# B&R Automation Studio project TD52 (part 131)

#### VisOPCyclic.st - Visualisation Communication Cyclic
```iecst
(*******************************************************************************
VisOP	 			 VISU and bus coupling variables

This code is confidential and proprietary to the INNIO Company.
It may not be used in any form, or reproduced in any manner,
without written permission of the INNIO Company.
Copyright, INNIO Company, 2023

Customized modifications: -
------------------------

History:
-------
V0.1.0	13.09.2012	Graus		new
V0.1.1	23.04.2013	Graus		MM2VIS.rP_Set_Min in AUTO and TEST to Para-value, otherwise is 0
V4.00.0 11.02.2014 	Graus,		change Version TO 4.0
V4.00.1	19.02.2014 zengerer		iIdx_OMSS, iIdx_RSS changed to DINT because of OPC UA troubles
V4.00.2 05.03.2014 	Graus,		add progress indication OF engine operation FOR VIS (iSt_VIS_Porgress)
V4.00.3 14.03.2014 	Graus,		add bEng_Rdy_Aut to MM2VIS structure and assign it for visualization
V4.01.0 19.05.2014  Denk		IN_OP.rP_RedDI_EU_Norm changed
V4.02.0 02.07.2014  Graus,		add MM2VIS.bP_Red_Sp_Lim1Act, 2 and 3
V4.02.1	15.10.2014	Caks,		added glow ignition power reduction
V4.02.2	17.02.2015	Graus,		add visu interface for power reduction by hierarchy controller
V4.02.3	04.05.2015	Denk,		add visu interfaces for OPC
V4.04.0	08.07.2016	Zengerer	BETA: Step Time Display Information
		17.11.2016	Gomez Ortiz	Addition of B2168 generator air inlet temperature power reduction
		21.12.2016  Denk		Modification for WinMOD simulation
V4.05.0 14.06.2017	Gomez Ortiz Addition of power limitation due to low engine cooling water temperature, Spec_Start_Load_release_manual_start.doc
V4.05.0 19.10.2017  Gomez Ortiz Addition of bImp_UnitOpHour to the MM2VIS struct
		24.10.2017	Zingerle	SWAT 920 Rel.5, power reduction with difference pressure minimum
		21.01.2018	Perktold,	hardware operation mode switch added
V4.07.0	11.10.2018	lettenb.	Di: tF_N_DI_Inc/Dec added for diagnosis
V4.07.4	29.03.2019	Hohensinner	Bugfixing: added missing interface to VIS for PRed CppInt
		26.04.2019	Hohensinner	Set minimum time for speed pulses for HMI to 2sec
V4.10.0 10.12.2020  Zuschnig	Included power reduction for Tecjet differential pressure
		18.01.2021	Perktold	included spec. gas p.red in MM2VIS
		25.01.2021	Zuschnig	Change MM2VIS.P_UNRED from Norm to kW
V4.11.0	20.08.2021 	Keller		Add Messages bMsg9057 - bMsg9060
		22.11.2021	Perktold,	added myPlant Remote Status computation
		22.12.2021	Andre		added Power reduction by CAN communication failure for half or more SAFI or too many SAFI reboots
V4.12.0	12.01.2023	Tinello		Deleted power reduction by T1HP / Added power reduction by T2HP and T2LP
		22.01.2023  Zuschnig	Include power reduction H2 content
		24.03.2023	Perktold	Write on PRed-MM2VIS variables just when ParaSetupOk is true - mitigation for wrong values on HMI
V4.13.0	05.07.2023	Zuschnig	Removed Step Time Display Information
  		26.01.2024 	Zuschnig 	Split of power reduction FPR

Instructions for use:
--------------------

Outstandings:
------------

(*******************************************************************************)

PROGRAM _CYCLIC

	(* Output: MM2VIS *)
	(* myPlant Remote Status computation *)
	IF bParaSetupOk_2s AND NOT bGnlTrip AND NOT bRequest_Bloc AND NOT OUT_OP.bEng_Bloc AND bOMSS_AUTO AND bRSS_REM AND (IN_OP.iIdx_SyOMSS = 2) AND Para.bRemoteReqMyPlantActive THEN
		MM2VIS.iMyPlant_Remote_Ready		:= 2;
	ELSE
		(* Reset myPlant demand in following cases, trip, engine blocking active, engine not in AUTO + REMOTE mode or function not active*)
		IF VIS2MM.bRemoteReq_myPlant THEN
			VIS2MM.bRemoteReq_myPlant 		:= FALSE;
		END_IF;
		IF Para.bRemoteReqMyPlantActive THEN
			MM2VIS.iMyPlant_Remote_Ready	:= 1;
		ELSE
			MM2VIS.iMyPlant_Remote_Ready	:= 0;
		END_IF;
	END_IF;

	MM2VIS.M_ANF := 			M_ANF;
	MM2VIS.iSt_OpMode_Main := 	iSt_OpMode_Main;
	MM2VIS.rN_Set := 			OUT_OP.rN_Set_Norm * Para.rN_EngNom;
	MM2VIS.rP_Act_Filt := 		OUT_OP.rP_Act_Norm_Filt * OUT_OP.rP_Nom;
	MM2VIS.rP_Set := 			OUT_OP.rP_Set_Norm * OUT_OP.rP_Nom;
	MM2VIS.P_UNRED := 			OUT_OP.rP_Set_Unred_Norm * OUT_OP.rP_Nom;

	MM2VIS.bP_Red_Active := 	OUT_OP.bP_Red_Active OR xTP_bP_Red_Active.Q;
	xTP_bP_Red_Active(IN := 	MM2VIS.bP_Red_Active, PT := T#1s);				(*min 1s TRUE to mitigate wrong values on HMI*)

	MM2VIS.RedPower := 			RedPower_Norm * OUT_OP.rP_Nom;
	MM2VIS.iIdx_Eng_State := 	iIdx_Eng_State;
	MM2VIS.iIdx_Pred_Type := 	OUT_OP.iIdx_Pred_Type;
	MM2VIS.iSt_OpMode_Sub := 	iSt_OpMode_Sub;
	MM2VIS.iSt_OpMode_Deg := 	iSt_OpMode_Deg;
	MM2VIS.bMsg2125 := 		bMsg2125;
	MM2VIS.bMsg2126 := 		bMsg2126;
	MM2VIS.bMsg2127 := 		bMsg2127;
	MM2VIS.bMsg2128 := 		bMsg2128;
	MM2VIS.bMsg2129 := 		bMsg2129;
	MM2VIS.bMsg2130 := 		bMsg2130;
	MM2VIS.bMsg2131 := 		bMsg2131;
	MM2VIS.bMsg2132 := 		bMsg2132;
	MM2VIS.bMsg2143 := 		bMsg2143;
	MM2VIS.bMsg2144 := 		bMsg2144;
	MM2VIS.bMsg2146 := 		bMsg2146;
	MM2VIS.bMsg2147 := 		bMsg2147;
	MM2VIS.bMsg2148 := 		bMsg2148;
	MM2VIS.bMsg2149 := 		bMsg2149;
	MM2VIS.bMsg2150 := 		bMsg2150;
	MM2VIS.bMsg2152 := 		bMsg2152;
	MM2VIS.bMsg2153 :=		bMsg2153;
	MM2VIS.bMsg2154 :=		bMsg2154;
	MM2VIS.bMsg2155 :=		bMsg2155;
	MM2VIS.bMsg2158 :=		bMsg2158;
	MM2VIS.bMsg2159 :=		bMsg2159;
	MM2VIS.bMsg2160 :=		bMsg2160;
	MM2VIS.bMsg2161 :=		bMsg2161;
	MM2VIS.bMsg2163 :=		bMsg2163;
	MM2VIS.bMsg2164 :=		bMsg2164;
	MM2VIS.bMsg2803 :=		bMsg2803;
	MM2VIS.bMsg3229 :=		bMsg3229;
	MM2VIS.bMsg3230 :=		bMsg3230;
	MM2VIS.bMsg3231 :=		bMsg3231;
	MM2VIS.bMsg2140 :=		bMsg2140;
	MM2VIS.bMsg3506 :=		bMsg3506;
	MM2VIS.bMsg2082 :=		bMsg2082;
	MM2VIS.bMsg1188 :=		bMsg1188;
	MM2VIS.bMsg2097 :=		bMsg2097;
	MM2VIS.bMsg1108 :=		bMsg1108;
	MM2VIS.bEng_RPSDem :=		OUT_OP.bEng_RPSDem;
	MM2VIS.bEng_Rdy_Aut_Exc :=	OUT_OP.bEng_Rdy_Aut_Exc;
	MM2VIS.rP_Ramp_IncGrad_All_Norm := OUT_OP.rP_Ramp_IncGrad_All_Norm;
	MM2VIS.rP_Ramp_DecGrad_All_Norm := OUT_OP.rP_Ramp_DecGrad_All_Norm;

	MM2VIS.bMsg1225 :=	bMsg1225;
	MM2VIS.bMsg1226 :=	bMsg1226;
	MM2VIS.bMsg1227 :=	bMsg1227;
	MM2VIS.bMsg1228 :=	bMsg1228;
	MM2VIS.bMsg1229 :=	bMsg1229;
	MM2VIS.bMsg1230 :=	bMsg1230;
	MM2VIS.bMsg1231 :=	bMsg1231;
	MM2VIS.bMsg1232 :=	bMsg1232;
	MM2VIS.bMsg1233 :=	bMsg1233;
	MM2VIS.bMsg1234 :=	bMsg1234;
	MM2VIS.bMsg1237 :=	bMsg1237;
	MM2VIS.bMsg1238 :=	bMsg1238;
	MM2VIS.bMsg1241 :=	bMsg1241;
	MM2VIS.bMsg1242 :=	bMsg1242;
	MM2VIS.bMsg1243 :=	bMsg1243;
	MM2VIS.bMsg1244 :=	bMsg1244;

	MM2VIS.bMsg2170 :=	bMsg2170;
	MM2VIS.bMsg2936 :=	bMsg2936;

	(* from HAL IO *)
	(* to HAL IO *)
	MM2VIS.bEng_Aux_Dem_CDR :=	OUT_OP.tEng_Aux_Dem_CDR.Do;
	MM2VIS.bEng_Run :=			OUT_OP.tEng_Run.Do;

	(* Input: VIS2MM *)
	bStart := 			VIS2MM.bStart;
	VIS2MM.bStart := 	FALSE;	(* reset VIS button *)
	bStop := 			VIS2MM.bStop;
	VIS2MM.bStop := 	FALSE;	(* reset VIS button *)

	(* HARDWARE OPERATION MODE SWITCHES *)
	IF IN_OP.tHW_Switches.bGoodQual THEN
		OUT_OP.iIdx_OMSS			:= IN_OP.tHW_Switches.iIdx_OMS_Hw;
		OUT_OP.iIdx_RSS 			:= IN_OP.tHW_Switches.iIdx_RMS_Hw;
		VIS2MM.iIdx_OMSS			:= INT_TO_DINT(IN_OP.tHW_Switches.iIdx_OMS_Hw);
		VIS2MM.iIdx_RSS				:= INT_TO_DINT(IN_OP.tHW_Switches.iIdx_RMS_Hw);
		MM2VIS.bDont_show_switches	:= TRUE;	(* DON'T show switches on HMI *)
	ELSE	(* OPERATION MODE SWITCHES ON HMI *)
		OUT_OP.iIdx_OMSS 			:= DINT_TO_INT(VIS2MM.iIdx_OMSS);
		OUT_OP.iIdx_RSS 			:= DINT_TO_INT(VIS2MM.iIdx_RSS);
		MM2VIS.bDont_show_switches	:= FALSE;	(* show switches on HMI *)
	END_IF;

	OUT_OP.bStart	:= 	bStart;		(* to AuxiliariesGeneral starter tasks *)
	OUT_OP.bStop	:= 	bStop;		(* to AuxiliariesGeneral starter tasks *)

	MM2VIS.bMainMode_Idle := xOpMode.Idle;
	MM2VIS.bMainMode_Grid := xOpMode.NetP;
	MM2VIS.bMainMode_Island := xOpMode.Island;

	xTON_ParaOK_1s(IN := IN_OP.tPB2MM.bParaSetupOk, PT := T#1s);	(*Delay to mitigate wrong values on HMI*)
	IF xTON_ParaOK_1s.Q THEN

		MM2VIS.rP_Nom			:=		OUT_OP.rP_Nom;

		MM2VIS.rP_RedDelta_Knck_Norm		:= 1.0 - IN_OP.rP_Red_Knck_Norm;
		MM2VIS.rP_RedDelta_Ch_T2s_Norm		:= 1.0 - IN_OP.rP_Red_Ch_T2s_Norm_TC5;
		MM2VIS.rP_RedDelta_Misf_Norm		:= 1.0 - IN_OP.rP_Red_Misf_Norm;
		MM2VIS.rP_RedDelta_EGT_Norm			:= 1.0 - IN_OP.rP_Red_EGT_Norm;
		MM2VIS.rP_RedDelta_T_InAirER_Norm	:= 1.0 - IN_OP.rP_Red_T_InAirER_Norm;
		MM2VIS.rP_RedDelta_Leanox_Norm		:= 1.0 - IN_OP.rP_Red_Leanox_Norm;
		MM2VIS.rP_RedDelta_CH4_Norm			:= 1.0 - IN_OP.rP_Red_CH4_Norm;
		MM2VIS.rP_RedDelta_GasPr_Norm		:= 1.0 - IN_OP.rP_Red_GasPr_Norm;
		MM2VIS.rP_RedDelta_SuctPr_Norm		:= 1.0 - IN_OP.rP_Red_SuctPr_Norm;
		MM2VIS.rP_RedDelta_TC_Norm			:= 1.0 - IN_OP.rP_Red_TC_Norm;
		MM2VIS.rP_RedDelta_T_HWR_Norm		:= 1.0 - IN_OP.rP_Red_T_HWR_Norm;
		MM2VIS.rP_RedDelta_T_ECW_Norm		:= 1.0 - IN_OP.rP_Red_T_ECW_Norm;
		MM2VIS.rP_RedDelta_T_Oil_Norm		:= 1.0 - IN_OP.rP_Red_T_Oil_Norm;
		MM2VIS.rP_RedDelta_Pr_PCGT_Norm		:= 1.0 - IN_OP.rP_Red_Pr_PCGT_Norm;
		MM2VIS.rP_RedDelta_CosPCtr_U_Norm 	:= 1.0 - IN_OP.rP_Red_CosPCtr_U_Norm;
		MM2VIS.rP_RedDelta_CosPCtr_F_Norm 	:= 1.0 - IN_OP.rP_Red_CosPCtr_F_Norm;
		MM2VIS.rP_RedDelta_CosPCtr_T_Norm 	:= 1.0 - IN_OP.rP_Red_CosPCtr_T_Norm;
		MM2VIS.rP_RedDelta_Sp_Lim1_Norm		:= 1.0 - IN_OP.rP_Red_Sp_Lim1_Norm;
		MM2VIS.rP_RedDelta_Sp_Lim2_Norm		:= 1.0 - IN_OP.rP_Red_Sp_Lim2_Norm;
		MM2VIS.rP_RedDelta_Sp_Lim3_Norm		:= 1.0 - IN_OP.rP_Red_Sp_Lim3_Norm;
		MM2VIS.rP_RedDelta_EVU_Norm			:= 1.0 - IN_OP.rP_RedDI_EU_Norm;
		MM2VIS.rP_RedDelta_AI_Norm			:= 1.0 - IN_OP.rP_Red_AI_Norm;
		MM2VIS.rP_RedDelta_ExtBus_Norm		:= 1.0 - IN_OP.rP_Red_ExtBus_Norm;
		MM2VIS.rP_RedDelta_Hum_Norm			:= 1.0 - IN_OP.rP_Red_Hum_Norm;
		MM2VIS.rP_RedDelta_PBC_Norm 		:= 1.0 - IN_OP.rP_Red_PBC_Norm;
		MM2VIS.rP_RedDelta_Knck_Opti_Norm	:= 1.0 - IN_OP.rP_Red_Knck_Opti_Norm;
		MM2VIS.rP_RedDelta_SG_Norm			:= 1.0 - MIN(IN_OP.rP_Red_SG_Norm_Pred, IN_OP.rP_Red_SG_Norm_FPR);
		MM2VIS.rP_RedDelta_Pr_CC_Norm		:= 1.0 - IN_OP.rP_Red_Pr_CC_Norm;
		MM2VIS.rP_RedDelta_HiCtr_Norm		:= 1.0 - IN_OP.rP_Red_HiCtr_Norm;
		MM2VIS.rP_RedDelta_T_Transformer_Norm		:= 1.0 - IN_OP.rP_Red_TransformerWarning_Norm;
		MM2VIS.rP_RedDelta_T_GenSwitchCab_Norm		:= 1.0 - IN_OP.rP_Red_TempMax_GenCB_Norm;
		MM2VIS.rP_RedDelta_T_GenAirIn_Norm	:= 1.0 - IN_OP.rP_Red_T_GenAirIn_Norm;
		MM2VIS.rP_RedDelta_Pr_GR_Norm		:= 1.0 - IN_OP.rP_Red_Pr_GR_Norm;
		MM2VIS.rP_RedDelta_CppInt_Norm		:= 1.0 - IN_OP.rP_Red_CppInt_Norm;
		MM2VIS.rP_RedDelta_CV_Norm			:= 1.0 - IN_OP.rP_Red_CV_Norm;
		MM2VIS.rP_RedDelta_Eta_Gen_Norm		:= 1.0 - IN_OP.rP_Red_Eta_Gen_Norm;
		MM2VIS.rP_RedDelta_SAErr_Norm		:= 1.0 - IN_OP.rP_Red_SAErr_Norm;
		MM2VIS.rP_RedDelta_SG_Norm			:= 1.0 - MIN(IN_OP.rP_Red_SG_Norm_Pred, IN_OP.rP_Red_SG_Norm_FPR);
		MM2VIS.rP_RedDelta_DPr_TJ_Norm		:= 1.0 - IN_OP.rP_Red_TJDiffPr_Norm;
		MM2VIS.rP_RedDelta_Ch_T2HP_Norm		:= 1.0 - IN_OP.rP_Red_Ch_T2HP_Norm;
		MM2VIS.rP_RedDelta_Ch_T2LP_Norm		:= 1.0 - IN_OP.rP_Red_Ch_T2LP_Norm;
		MM2VIS.rP_RedDelta_H2_Norm			:= 1.0 - IN_OP.rP_Red_H2_Norm;
	END_IF;

	xTON_ParaOK_2s(IN := IN_OP.tPB2MM.bParaSetupOk, PT := T#2s);		(*Delay to mitigate wrong values on HMI*)
	IF xTON_ParaOK_2s.Q THEN

		MM2VIS.rP_Red_EGT		:=		IN_OP.rP_Red_EGT_Norm	*	OUT_OP.rP_Nom;
		MM2VIS.rP_Red_Misf		:=		IN_OP.rP_Red_Misf_Norm	*	OUT_OP.rP_Nom;
		MM2VIS.rP_Red_Leanox	:=		IN_OP.rP_Red_Leanox_Norm *	OUT_OP.rP_Nom;
		MM2VIS.rP_Red_CH4		:=		IN_OP.rP_Red_CH4_Norm	*	OUT_OP.rP_Nom;
		MM2VIS.rP_Red_EVU		:=		IN_OP.rP_RedDI_EU_Norm	*	OUT_OP.rP_Nom;
		MM2VIS.rP_Red_GasPr		:=		IN_OP.rP_Red_GasPr_Norm	*	OUT_OP.rP_Nom;
		MM2VIS.rP_Red_SuctPr	:=		IN_OP.rP_Red_SuctPr_Norm *	OUT_OP.rP_Nom;
		MM2VIS.rP_Red_AI		:=		IN_OP.rP_Red_AI_Norm	*	OUT_OP.rP_Nom;
		MM2VIS.rP_Red_CosPCtr_F	:=		IN_OP.rP_Red_CosPCtr_F_Norm	*	OUT_OP.rP_Nom;
		MM2VIS.rP_Red_CosPCtr_U	:=		IN_OP.rP_Red_CosPCtr_U_Norm	*	OUT_OP.rP_Nom;
		MM2VIS.rP_Red_CosPCtr_T	:=		IN_OP.rP_Red_CosPCtr_T_Norm	*	OUT_OP.rP_Nom;
		MM2VIS.rP_Red_TC		:=		IN_OP.rP_Red_TC_Norm	*	OUT_OP.rP_Nom;
		MM2VIS.rP_Red_Sp_Lim1	:=		IN_OP.rP_Red_Sp_Lim1_Norm	*	OUT_OP.rP_Nom;
		MM2VIS.rP_Red_Sp_Lim2	:=		IN_OP.rP_Red_Sp_Lim2_Norm	*	OUT_OP.rP_Nom;
		MM2VIS.rP_Red_Sp_Lim3	:=		IN_OP.rP_Red_Sp_Lim3_Norm	*	OUT_OP.rP_Nom;
		MM2VIS.rP_Red_Knck		:=		IN_OP.rP_Red_Knck_Norm	*	OUT_OP.rP_Nom;
		MM2VIS.rP_Red_Ch_T2s	:=		IN_OP.rP_Red_Ch_T2s_Norm_TC5	*	OUT_OP.rP_Nom;
		MM2VIS.rP_Red_T_HWR		:=		IN_OP.rP_Red_T_HWR_Norm	*	OUT_OP.rP_Nom;
		MM2VIS.rP_Red_T_ECW		:=		IN_OP.rP_Red_T_ECW_Norm	*	OUT_OP.rP_Nom;
		MM2VIS.rP_Red_T_Oil		:=		IN_OP.rP_Red_T_Oil_Norm	*	OUT_OP.rP_Nom;
		MM2VIS.rP_Red_Pr_PCGT	:=		IN_OP.rP_Red_Pr_PCGT_Norm *	OUT_OP.rP_Nom;
		MM2VIS.rP_Red_ExtBus	:=		IN_OP.rP_Red_ExtBus_Norm *	OUT_OP.rP_Nom;
		MM2VIS.rP_Red_T_InAirER	:=		IN_OP.rP_Red_T_InAirER_Norm	*	OUT_OP.rP_Nom;
		MM2VIS.rP_Red_Hum		:= 		IN_OP.rP_Red_Hum_Norm	*	OUT_OP.rP_Nom;
		MM2VIS.rP_Red_PBC		:= 		IN_OP.rP_Red_PBC_Norm	*	OUT_OP.rP_Nom;
		MM2VIS.rP_Red_Knck_Opti	:= 		IN_OP.rP_Red_Knck_Opti_Norm	*	OUT_OP.rP_Nom;
		MM2VIS.rP_Red_SG		:= 		MIN(IN_OP.rP_Red_SG_Norm_Pred, IN_OP.rP_Red_SG_Norm_FPR) * OUT_OP.rP_Nom;
		MM2VIS.rP_Red_Pr_CC		:=		IN_OP.rP_Red_Pr_CC_Norm	*	OUT_OP.rP_Nom;
		MM2VIS.rP_Red_HiCtr		:=		IN_OP.rP_Red_HiCtr_Norm	*	OUT_OP.rP_Nom;
		MM2VIS.rP_Red_T_Transformer		:=	IN_OP.rP_Red_TransformerWarning_Norm	*	OUT_OP.rP_Nom;
		MM2VIS.rP_Red_T_GenSwitchCab	:=	IN_OP.rP_Red_TempMax_GenCB_Norm	*	OUT_OP.rP_Nom;
		MM2VIS.rP_Red_T_GenAirIn	:=	IN_OP.rP_Red_T_GenAirIn_Norm	*	OUT_OP.rP_Nom;
		MM2VIS.bP_Red_Sp_Lim1Act	:= 	IN_OP.bP_Red_Sp_Lim1Act;
		MM2VIS.bP_Red_Sp_Lim2Act	:= 	IN_OP.bP_Red_Sp_Lim2Act;
		MM2VIS.bP_Red_Sp_Lim3Act	:= 	IN_OP.bP_Red_Sp_Lim3Act;
		MM2VIS.rP_Red_Pr_GR			:= 	IN_OP.rP_Red_Pr_GR_Norm	*	OUT_OP.rP_Nom;
		MM2VIS.rP_Red_CppInt		:= 	IN_OP.rP_Red_CppInt_Norm	*	OUT_OP.rP_Nom;
		MM2VIS.rP_Red_CV			:= 	IN_OP.rP_Red_CV_Norm	*	OUT_OP.rP_Nom;
		MM2VIS.rP_Red_Eta_Gen		:=	IN_OP.rP_Red_Eta_Gen_Norm	*	OUT_OP.rP_Nom;
		MM2VIS.rP_Red_SAErr			:=	IN_OP.rP_Red_SAErr_Norm	*	OUT_OP.rP_Nom;
		MM2VIS.rP_Red_SG_Norm		:=	MIN(IN_OP.rP_Red_SG_Norm_Pred, IN_OP.rP_Red_SG_Norm_FPR) * OUT_OP.rP_Nom;
		MM2VIS.rP_Red_DPr_TJ		:= 	IN_OP.rP_Red_TJDiffPr_Norm	*	OUT_OP.rP_Nom;
		MM2VIS.rP_Red_H2			:= 	IN_OP.rP_Red_H2_Norm	*	OUT_OP.rP_Nom;
		MM2VIS.rP_Red_Ch_T2HP		:=	IN_OP.rP_Red_Ch_T2HP_Norm *	OUT_OP.rP_Nom;
		MM2VIS.rP_Red_Ch_T2LP		:=	IN_OP.rP_Red_Ch_T2LP_Norm *	OUT_OP.rP_Nom;

		IF (OUT_OP.iIdx_OMSS = 2)(*AUTO*) OR (OUT_OP.iIdx_OMSS = 3)(*TEST*) THEN
			MM2VIS.rP_Set_Min	:=		OUT_OP.rP_Set_Min_Norm	*	OUT_OP.rP_Nom;
		ELSE
			MM2VIS.rP_Set_Min	:= 		0;
		END_IF;
	END_IF;

	MM2VIS.bMsg2122 :=	bMsg2122;
	MM2VIS.bMsg2123 :=	bMsg2123;
	MM2VIS.bMsg2124 :=	bMsg2124;
	MM2VIS.bMsg2133 :=	bMsg2133;
	MM2VIS.bMsg2134 :=	bMsg2134;
	MM2VIS.bMsg2135 :=	bMsg2135;
	MM2VIS.bMsg2136 :=	bMsg2136;
	MM2VIS.bMsg2137 :=	bMsg2137;
	MM2VIS.bMsg2138 :=	bMsg2138;
	MM2VIS.bMsg2813 :=	bMsg2813;
	MM2VIS.bMsg9057 := 	bIsland_NoffsCust;	(* B9057 - Isolated operation - external speed reference mode *)
	MM2VIS.bMsg9058 := 	bPset_Droop_Bus;	(* B9058 - message power setpoint by Bus input Droop *)
	MM2VIS.bMsg9059 := 	bPset_Droop_AI;		(* B9059 - message power setpoint by analog input Droop *)
	MM2VIS.bMsg9060 := 	bPset_Droop_Man;	(* B9060 - message power setpoint by internal HMI value Droop *)

	IF (OUT_OP.rP_Act_Norm >=0.95) THEN (* The engine operates at 95% load or higher *)
		MM2VIS.iSt_VIS_Porgress := 6;
	ELSIF IN_OP.bLeanox_Active THEN		(* leanox controller activatd *)
		MM2VIS.iSt_VIS_Porgress := 5;
	ELSIF xOpMode.NetP OR xOpMode.Island THEN (* mains parallel or isolated operation mode *)
		MM2VIS.iSt_VIS_Porgress := 4;
	ELSIF xOpMode.Idle THEN				(* idle mode *)
		MM2VIS.iSt_VIS_Porgress := 3;
	ELSIF (iIdx_Eng_State = 10) THEN	(* engine start up *)
		MM2VIS.iSt_VIS_Porgress := 2;
	ELSIF (M_ANF = TRUE) THEN			(* module has been activated *)
		MM2VIS.iSt_VIS_Porgress := 1;
	ELSE								(* module has not been activated *)
		MM2VIS.iSt_VIS_Porgress := 0;
	END_IF

	MM2VIS.bEng_Rdy_Aut := OUT_OP.bEng_Rdy_Aut;
	MM2VIS.bEng_Rdy_Rem := OUT_OP.tEng_Rdy_Rem.Do;
	MM2VIS.bEng_Aux_Dem := OUT_OP.bEng_Aux_Dem;
	MM2VIS.bImp_OpHour  := OUT_OP.tImp_OpHour.Do;
	MM2VIS.bImp_UnitOpHour  := OUT_OP.bImp_UnitOpHour;
	MM2VIS.bImp_Start	:= OUT_OP.bImp_Start;

	xTP_F_N_DI_Inc(IN:= EDGEPOS(IN_OP.tF_N_DI_Inc.Di), PT:= T#2s);	(* DI synch.increase speed *)
	MM2VIS.bF_N_DI_Inc		:= xTP_F_N_DI_Inc.Q;

	xTP_F_N_DI_Dec(IN:= EDGEPOS(IN_OP.tF_N_DI_Dec.Di), PT:= T#2s);	(* DI synch.decrease speed *)
	MM2VIS.bF_N_DI_Dec		:= xTP_F_N_DI_Dec.Q;

END_PROGRAM
```

#### VisOPInit.st - Visualisation Communication Init
```iecst
(********************************************************************
 * COPYRIGHT -- INNIO Company
 ********************************************************************
 * Program: VisOP
 * File: VisOPInit.st
 * Author: 105051472
 * Created: September 13, 2012
 ********************************************************************
 * Implementation of program VisOP
 ********************************************************************)

PROGRAM _INIT

END_PROGRAM
```

#### VisOP.var - Local variables
```iecst
(********************************************************************
 * COPYRIGHT -- INNIO Company
 ********************************************************************
 * Program: VisOP
 * File: VisOP.var
 * Author: 105051472
 * Created: September 13, 2012
 ********************************************************************
 * Local variables of program VisOP
 ********************************************************************)
VAR
	xTP_F_N_DI_Inc : TP;
	xTP_F_N_DI_Dec : TP;
	xTON_ParaOK_1s : TON;
	xTON_ParaOK_2s : TON;
	xTP_bP_Red_Active : TP;
END_VAR
```

### Program Logical/Opstate/ParOP (IEC) - + Parameter Management OpState

- perm_par.st (not readable text: treated as protected, skipped)

#### perm_par.var
```iecst
VAR
	tParaIntern : ParaHandler_typ; (*Connector type to perm_par*)
	tMM2ParaBase_ReadBack : MM2ParaBase_type; (*INTERNAL! V4.06 new readback structure for information from previous tasks*)
	bWriteDataObj : BOOL; (* TRUE=write data object module *)
	bDataObjLenErr : BOOL; (*Error occured in permem: data module size missmatch*)
	bCreateDataObj : BOOL; (* TRUE=create new data object *)
	bWriteOnce : BOOL; (* write permanent memory once *)
	DatObjCreate_01 : DatObjCreate; (* data object create *)
	DatObjInfoBak_02 : DatObjInfo; (* data object info *)
	DatObjDelete_01 : DatObjDelete; (* data object delete *)
	DatObjRead_01 : DatObjRead; (* data object read *)
	DatObjRead_02 : DatObjRead; (* manual initiated data object read *)
	DatObjWrite_01 : DatObjWrite; (* data object write *)
	DatObjDelete_02 : DatObjDelete; (* data object delete *)
	DatObjDelete_11 : DatObjDelete; (*Delete Backup File*)
	DatObjInfo_01 : DatObjInfo; (* data object info *)
	DatObjInfo_02 : DatObjInfo; (* data object info *)
	szModuleName : STRING[35]; (* module name of object *)
	szModuleNameBackup : STRING[35]; (* module name of posiibly created backup object *)
	DatObjCopy_01 : DatObjCopy;
	bCopyDataObj : BOOL;
	TON_WarnDelay : TON;
	TON_WritePMEM : TON; (* delay write permanent memory *)
	ulPMPointer : UDINT; (* adress of actual checksum value *)
	ulChecksum : UDINT; (* parameter checksum value *)
	pm_len : UDINT; (* permanent value lenght *)
	ulChecksumOld : UDINT; (* last vlaue of parameter checksum *)
	ulChkValue : UDINT; (* actual value of parameter pointer *)
	pm_id : UDINT; (* permanent value identifier *)
	pm_p : UDINT; (* permanent value pointer *)
	DatObjInfo_META : DatObjInfo;
	DatObjRead_META : DatObjRead;
	szMetaDataRaw : STRING[2000];
	szMetaData : ARRAY[0..4] OF STRING[35];
	szMetaDataVis : ARRAY[0..3] OF STRING[35];
	ssIndex : INT;
	ssCount : INT;
	ucMetaDataRaw : ARRAY[0..2000] OF USINT;
	ssCount2 : INT;
	szMetaDataFile : STRING[10];
	szText1 : STRING[20];
	pv_adr_IN_XX_tPB2MM : UDINT;
	pv_lng : UDINT;
	pv_lng_IN_XX_tPB2MM : UDINT;
	pv_lng_OUT_XX_tPB2MM : UDINT;
	szText2 : STRING[20];
	pv_adr_OUT_XX_tXX2PB : UDINT;
END_VAR
VAR CONSTANT
	ERR_NOERROR : UINT := 0;
END_VAR
VAR
	usPMWriteCnt : UINT;
	pm_Error : UDINT; (* permanent value error *) (* Deleted: pm : ParaMem_typ; permanent memory tags mathias, 22.8.11*)
	fun_Error : UDINT := 0; (*state > 0 = function error*)
	xLocalParaCheck : ParaCheckFUB; (*local function instance to check parameter values*)
	TON_ParaSetupOk : TON;
	bParaCheckSystemOk : BOOL;
	iDebug_ParaOkChecked : UDINT;
	bRestoreBackupDataObj : BOOL := FALSE;
	bRestoreDataObjContent : BOOL := FALSE;
	pm_id_backup : UDINT;
	pm_p_Backup : UDINT;
	DatObjCopy_02 : DatObjCopy;
	bDeleteBackupDataObj : BOOL := FALSE; (*Command to delete backup data module file on purpose*)
	bDebugPara : ARRAY[0..5] OF BOOL;
	ssIndex2 : INT;
	ssIndex3 : INT;
	ssIndex4 : INT;
	ssIndexVis : INT;
	szText : STRING[40];
	pv_adr_Para : UDINT;
	szParaSnippet : ARRAY[0..5] OF STRING[150];
	szParaIndex : STRING[10];
	slValue : DINT;
	iModuleDLD_ResetCount : INT;
	bDownloadDetected : BOOL;
	bFlagParaStructCopyWorking : BOOL; (*true, if cyclic para copying is active, 1 false cycle at every copy *)
	bStoreInitParaInDataObj : BOOL := FALSE;
	bTestflag : BOOL;
	bReadOutMETA_Once : BOOL;
	tParaCheck_iPvAdress : ARRAY[0..5] OF UDINT;
	tParaCheck_iPvLengt : ARRAY[0..5] OF UDINT;
	tParaCheck_rPvValue : ARRAY[0..5] OF REAL;
	tParaCheck_rRangeMIN : ARRAY[0..5] OF REAL;
	tParaCheck_rRangeMAX : ARRAY[0..5] OF REAL;
	tParaCheck_szPvName : ARRAY[0..5] OF STRING[35];
	ssFormatDetected : INT;
	szMetaDataPart : STRING[150];
	szFullTaskName : STRING[35];
	szFullMetaModuleName : STRING[35];
	debugLen : INT;
	debugSize : INT := 0;
	strcat_adr1 : UDINT;
	strcat_adr2 : UDINT;
	ssIndexTN : INT;
	bAlternate : BOOL;
	n : INT;
	iAlternateChecksum : DINT;
	iAlternateChecksumOld : DINT;
	ulDebugChkValue : ARRAY[0..999] OF UDINT;
	Adr1 : UDINT;
	Adr2 : UDINT;
	usPMWriteCntStepsize : UINT := 1; (*different step sizes to help debug*)
	usPMWriteCntXOR : UINT;
	usPMWriteCntAltSum : UINT;
	ulAdrPM : UDINT;
	usChkValuePM : USINT;
	ulAdrPara : UDINT;
	ulPara_len : UDINT;
	usChkValuePara : USINT;
	iDebugCountPMDifferences : DINT := 0;
	bEngineRunDetected : BOOL; (*detection status bit autocommand 100 /101  for engine run state*)
	ucMetaDataDebugInfoLine : ARRAY[0..24] OF STRING[80];
	ssIndexMand : INT := 0;
	szMetaDataMand : STRING[35];
	iMyErrorInfo_Autoreset : DINT; (*internal autoreset counter*)
	ssIndex_Version : INT; (*internal*)
	ssIndex_BU : INT; (*internal*)
	ssIndex_BU2 : INT; (*internal*)
END_VAR
```

### Program Logical/Opstate/default_OP (IEC) - OpState setting values

#### default_OPCyclic.st - OpState setting values
```iecst
(*******************************************************************************
default		value set

This code is confidential and proprietary to the INNIO Company.
It may not be used in any form, or reproduced in any manner,
without the express written permission of the INNIO Company.
Copyright, INNIO Company, 2019

Customized modifications: -
------------------------

History:
-------
V0.00.0	19.10.2012	Graus,		new
V4.00.0 11.02.2014 	Graus,		change Version TO 4.0
V4.00.0 17.11.2016 	Gwiggner,	change Version TO 4.04
		02.02.2017	lettenb.	OUT_OP.bEng_Bloc: ...FC_Rdy included(sky)
V4.07.0 03.12.2018	lettenb.	tScavVaClosed added, bugfix for option N2 scavenging without scav.flap
V4.10.0 03.08.2020	lettenb.	tScavFanCB_trip, tGenIF_CB_On added

Instructions for use:
--------------------
Outstandings:
------------
*******************************************************************************)
PROGRAM _CYCLIC

	(* default TRUE setting for not existing Di's *)
	IN_OP.tRel_MasCtr.Di		:=	IN_OP.tRel_MasCtr.Di		OR	NOT IN_OP.tRel_MasCtr.GoodQual;

	IN_OP.tScavFanFC_Rdy.Di		:=	IN_OP.tScavFanFC_Rdy.Di		OR	NOT IN_OP.tScavFanFC_Rdy.GoodQual;
	IN_OP.tECWP_FC_Rdy.Di		:=	IN_OP.tECWP_FC_Rdy.Di		OR	NOT IN_OP.tECWP_FC_Rdy.GoodQual;
	IN_OP.tEOP_FC_Rdy.Di		:=	IN_OP.tEOP_FC_Rdy.Di		OR	NOT IN_OP.tEOP_FC_Rdy.GoodQual;
	IN_OP.tBbBlower_FC_Rdy.Di	:=	IN_OP.tBbBlower_FC_Rdy.Di	OR	NOT IN_OP.tBbBlower_FC_Rdy.GoodQual;
	IN_OP.tScavVaClosed.Di		:=	IN_OP.tScavVaClosed.Di		OR	NOT IN_OP.tScavVaClosed.GoodQual;
	IN_OP.tScavFanCB_trip.Di	:=	IN_OP.tScavFanCB_trip.Di	OR	NOT	IN_OP.tScavFanCB_trip.GoodQual;
	IN_OP.tGenIF_CB_On.Di		:=	IN_OP.tGenIF_CB_On.Di		OR	NOT	IN_OP.tGenIF_CB_On.GoodQual;
	IN_OP.tECWP_CB_On.Di		:=	IN_OP.tECWP_CB_On.Di		OR	NOT	IN_OP.tECWP_CB_On.GoodQual;

END_PROGRAM
```

### Program Logical/Opstate/PermOP (IEC) - + Permanent variable storage OP

- perm_par.st (not readable text: treated as protected, skipped)

#### perm_par.var
```iecst
VAR
	tParaIntern : ParaHandler_typ; (*Connector type to perm_par*)
	bWriteDataObj : BOOL; (* TRUE=write data object module *)
	bDataObjLenErr : BOOL; (*Error occured in permem: data module size missmatch*)
	bCreateDataObj : BOOL; (* TRUE=create new data object *)
	write_once : BOOL; (* write permanent memory once *)
	DatObjCreate_01 : DatObjCreate; (* data object create *)
	DatObjInfo_01 : DatObjInfo; (* data object info *)
	DatObjRead_01 : DatObjRead; (* data object read *)
	DatObjWrite_01 : DatObjWrite; (* data object write *)
	ModuleName : STRING[35]; (* module name of object *)
	TON_WarnDelay : TON;
	TON_WritePMEM : TON; (* delay write permanent memory *)
	ulPMPointer : UDINT; (* adress of actual checksum value *)
	ulChecksum : UDINT; (* parameter checksum value *)
	pm_len : UDINT; (* permanent value lenght *)
	ulChecksumOld : UDINT; (* last vlaue of parameter checksum *)
	ulChkValue : UDINT; (* actual value of parameter pointer *)
	pm_id : UDINT; (* permanent value identifier *)
	pm_p : UDINT; (* permanent value pointer *)
	DatObjDelete_PermMem : DatObjDelete; (* delete data object *)
END_VAR
VAR CONSTANT
	ERR_NOERROR : UINT := 0;
END_VAR
VAR
	usPMWriteCnt : UINT;
	pm_Error : UINT; (* permanent value error *) (* Deleted: pm : ParaMem_typ; permanent memory tags mathias, 22.8.11*)
	xLocalParaCheck : ParaCheckFUB; (*local function instance to check parameter values*)
	Debug_pm_Error : UINT := 0;
	Debug_iPermStatus : DINT := 0;
END_VAR
```

### Package Logical/ParaBase - PB: Parameter Base

### Data object Logical/ParaBase/META_PB (Simple) - Simple data object.

#### META_PB.dat
```
; *******************************************************************************
; AGGR: Module Meta Data (data module)
;
; This code is confidential and proprietary to the INNIO Company.
; It may not be used in any form, or reproduced in any manner, without the express
; written permission of the INNIO Company.
; Copyright, INNIO Company, 2020
;
; Customized modifications: -
; ------------------------
;
; History:
; -------
; V3.99	  06-03-2013	Weitzer,	generated for modular software
; V3.99.1 29-05-2013	Zengerer	initial dependencies prepared
; V3.99.2 25-06-2013	Zengerer 	Prototype meta with function description
; V4.00.0 29-01-2014				release version, unchanged
; V4.13.1 14-03-2024	Zengerer 	version updated here - detailed change descriptions only inside tasks or in info section
;
; Instructions for use:
; --------------------
; make only changes at the version numbers
; OBEY XML FORMATING RULES!
;
; Outstandings:
; ------------
; datamodule syntax checker
; (caution: syntax errors here may cause plc runtime errors!)
;
; *******************************************************************************
;
"<META>"
;
; Module ID
"<MODUL>PB</MODUL>"
;
; Module Version (xx.yy.zz.cc)
"<VERSION>04.13.01.00</VERSION>"
;
; Module Basisupdate Version BU (00-99)
"<BASISUPDATE_VERSION='00' /BASISUPDATE_VERSION>"
;
; Optional: specify order number for limitated module usage
"<ORDER></ORDER>" ;<!--(optional for restricted customizations; missing statement makes module valid for all orders)-->
;
; Parameter Check <PARAn Name='aAbcdef' MIN='xxx' MAX='yyy' />  (watch for correct spacings and apostrophs!)
"<PARAMETER_CHK>"
"	<PARA1 Name='iEng_Motortype' MIN='208' MAX='920' />"
"	<PARA2 />"
"	<PARA3 />"
"	<PARA4 />"
"	<PARA5 />"
"</PARAMETER_CHK>"
;
; Statement, that this module´s parameter check passing is mandatory (PB is allways mandatory, so other statements than TRUE here in this module are not possible)
"<MANDATORYMODULE>TRUE</MANDATORYMODULE>"
;
; Permanent Datamodule Filenames<!-- enter filenames for counter and INTERNAL parameter only; filename without extention-->
"<DATAMODULES>" ;<!-- optional; mehrere DATAMODULES erlaubt-->
"	<DATAMODULE>par_PB</DATAMODULE>"
"	<DATAMODULE>perm_PB</DATAMODULE>"
"</DATAMODULES>"
;
; Dependencies Modules (MMxx.yy.zz.cc)
"<DEPENDENCIES>"
"	<DEPENDENCY MODULE='AB' VERSION='04.00.00.00' />"
"	<DEPENDENCY MODULE='HA' VERSION='04.10.00.00' />"
"	<DEPENDENCY MODULE='OP' VERSION='04.13.00.00' />"
"   <DEPENDENCY VISVERSION='02.14.00.00' />"			; Dependencies Visualization
"</DEPENDENCIES>"
;
; Module function description
"<MODULEFUNCTION>" ;<!-- short overview documentation of module function; add reference to detailed information, if available-->
"	<General>	"
"	It provides and forwards a collection of status information from the software modules for visualisation purposes and diagnosis. "
"	</General>	"
""
"	<F1 Name='Data collection' LastModified='4.0.0.0'>"
"	The module 'ParaBase' collects basically necessary status messages from all modules.	"
"	</F1>"
"	<F2 Name='Release Controller Operation' LastModified='4.0.0.0'>"
"	 Processes this information to detect system integrity, to release controller operation.	"
"	</F2>"
"	<F3 Name='Load and Save' LastModified='4.0.0.0'>"
"	Coordinates parameter load and save activities in all the modules ParXX- tasks.	"
"	</F3>"
"	<F4 Name='Update Info:' LastModified='4.4.1.0'>"
"	Bugfix 17.1.2014 in all the modules ParXX- tasks.	"
"   Support for Para.iParaBaseExtensionCommand 101 = bSendAutoCommands "
"	DatObjRead_META(enable =FALSE) clean up"
"	</F4>"
"	<F5 Name='PermStatus' LastModified='4.6.0.0'>"
"	Perm File Status NEEDS LIBRARY UPDATE ParaBase V4.06 2018-10-12 Ze	for extendet Type declaration for Perm Statusinfo"
"	</F5>"
"	<F6 Name='Perm File Status Info' LastModified='4.7.0.0'>"
"	Perm task handling with info collection structure for centralised para file status handling "
"	</F6>"
"	<F7 Name='PermCntCheck' LastModified='4.13.0.0'>"
"	Perm File sanity checks by OpHr counter value comparison 2023-05-24 Ze"
"	</F7>"
""
"	<Info>"
"	The ParXX- task in every module actualy does power fail resistant and download resistant parameter saving and handling for all the modules permanent parameter in its own 'Para.' Structure.	"
"	It allso provides the communication interface to the ParaBase Module.	"
"	</Info>"
""
"	<Customized LastModified='4.0.0.0'>	"
"	none "
"	</Customized>	"
""
"</MODULEFUNCTION>"
;
"</META>"
```

### ParaBase.typ - Package data types
```iecst
(********************************************************************
 * COPYRIGHT -- INNIO Company
 ********************************************************************
 * Package: ParaBase
 * File: ParaBase.typ
 * Author: zengeres
 * Created: September 14, 2012
 ********************************************************************
 * Data types of package ParaBase
 ********************************************************************)

TYPE
	IN_PB_Struct : 	STRUCT
		tVE2PB : MM2ParaBase_type; (*VE Ventilation*) (*OldName: new PV; Cycle: 5;*)
		tHC2PB : MM2ParaBase_type; (*HC Heating Cooling*) (*OldName: new PV; Cycle: 5;*)
		tEX2PB : MM2ParaBase_type; (*EX Exhaust*) (*OldName: new PV; Cycle: 5;*)
		tTR2PB : MM2ParaBase_type; (*TR ParaBase*) (*OldName: new PV; Cycle: 5;*)
		tGC2PB : MM2ParaBase_type; (*GC Generator Control*) (*OldName: new PV; Cycle: 5;*)
		tCU2PB : MM2ParaBase_type; (*CU Customized*) (*OldName: new PV; Cycle: 5;*)
		tMO2PB : MM2ParaBase_type; (*MO Monic*) (*OldName: new PV; Cycle: 5;*)
		tIC2PB : MM2ParaBase_type; (*IC ICxxx*) (*OldName: new PV; Cycle: 5;*)
		tIG2PB : MM2ParaBase_type; (*IG Ignition*) (*OldName: new PV; Cycle: 5;*)
		tSY2PB : MM2ParaBase_type; (*SY Synchronization*) (*OldName: new PV; Cycle: 5;*)
		tCP2PB : MM2ParaBase_type; (*CP Coupling*) (*OldName: new PV; Cycle: 5;*)
		tEC2PB : MM2ParaBase_type; (*EC EngineController*) (*OldName: new PV; Cycle: 5;*)
		tEG2PB : MM2ParaBase_type; (*EG EngineGeneral*) (*OldName: new PV; Cycle: 5;*)
		tEM2PB : MM2ParaBase_type; (*EM Exhaust Monitoring*) (*OldName: new PV; Cycle: 5;*)
		tKN2PB : MM2ParaBase_type; (*KN Knocking*) (*OldName: new PV; Cycle: 5;*)
		tGM2PB : MM2ParaBase_type; (*GM GasMixer*) (*OldName: new PV; Cycle: 5;*)
		tGR2PB : MM2ParaBase_type; (*GR Grid Codes*) (*OldName: new PV; Cycle: 5;*)
		tGT2PB : MM2ParaBase_type; (*GT GasTrain*) (*OldName: new PV; Cycle: 5;*)
		tAG2PB : MM2ParaBase_type; (*AG AuxiliariesGeneral*) (*OldName: new PV; Cycle: 5;*)
		tOP2PB : MM2ParaBase_type; (*OP Opstate*) (*OldName: new PV; Cycle: 5;*)
		tSA2PB : MM2ParaBase_type; (*SA SAFI*) (*OldName: new PV; Cycle: 5;*)
		tKL2PB : MM2ParaBase_type; (*KL KLS98*) (*OldName: new PV; Cycle: 5;*)
		tGD2PB : MM2ParaBase_type; (*GD Gas Dosing (Tecjet)  ALT: GMU	GasMeteringUnit*) (*OldName: new PV; Cycle: 5;*)
		tCH2PB : MM2ParaBase_type; (*CH ChargingUnit*) (*OldName: new PV; Cycle: 5;*)
		tHA2PB : MM2ParaBase_type; (*HA HalIO*) (*OldName: new PV; Cycle: 5;*)
		tAB2PB : MM2ParaBase_type; (*AB AlarmBase Vorsicht NAME ABWEICHEND wegen Konflikt mit Amm- RÜCKGÄNGIG GEMACHT*) (*OldName: new PV; Cycle: 5;*)
		tCB2PB : MM2ParaBase_type; (*prepared: CBM Module*) (*OldName: new PV; Cycle: 5;*)
		tVI2PB : MM2ParaBase_type; (*VI Visu*) (*OldName: new PV; Cycle: 5;*)
		tPB2PB : MM2ParaBase_type; (*INTERNAL USE ONLY in PB module! Selbstgespräche...*) (*OldName: new PV; Cycle: 5;*)
		tPB2MM : ParaBase2MM_type; (*INTERNAL USE ONLY  in PB module! Selbstgespräche wieder zurück...*) (*OldName: new PV; Cycle: 5;*)
		tTB2PB : MM2ParaBase_type; (*USE ONLY for TESTBENCH module!*) (*OldName: new PV; Cycle: 5;*)
		iPassLevel : INT; (*pass level actual*) (*OldName: Userlevel; Cycle: 5;*)
		tResetRemExt : HALioDi_Type; (*reset remote external*) (*OldName: new PV; Cycle: 5;*)
		tGCB_On : HALioDi_Type; (*generator circuit breaker closed*) (*OldName: GS_EIN; Cycle: 5;*)
		tGCB_RUC : HALioDo_Type; (*generator circuit breaker release undervoltage coil*) (*OldName: USP; Cycle: 5;*)
		tSafetyLoop_Eng : HALioDi_Type; (*safety loop engine*) (*OldName: new PV; Cycle: 5;*)
		iIdx_OMSS : INT; (*operation selection*) (*OldName: BWS_H, BWS_A, BHS_HA,; Cycle: 5;*)
		iSt_OpMode : UDINT; (*engine operation status*) (*OldName: verschiedene; Cycle: 5;*)
		rN_EngAct : REAL; (*engine speed actual [1/min]*) (*OldName: n_ist; Cycle: 5;*)
		iCnt_OpHours : DINT; (* engine operating hours counter (from Module Opstate)*) (*OldName:betrieb_h;Cycle:2;*)
		iCnt_Starts : DINT; (* start counter  (from Module Opstate)*) (*OldName:start_z;Cycle:2;*)
		iCnt_FastStarts : DINT; (*Fast  start counter  (from Module Opstate)*)
		iCnt_UnitOpHours : DINT; (* unit operating hours counter (from Module Opstate)*)
		StationIO : BOOL;
		bSimWinMOD_Active : BOOL; (*V4.10*)
		tAlarmB2PB : AmmBase2MM; (* OWN AlarmBase CONNECTOR as Ammm- Structuretype*) (*OldName: new PV; Cycle: 5;*)
	END_STRUCT;
	OUT_PB_Struct : 	STRUCT
		iCnt_OpHours_Set : DINT; (*new V4.13 for ParaBase Counter Set*)
		iCnt_UnitOpHours_Set : DINT; (*new V4.13 for ParaBase Counter Set*)
		iCnt_Starts_Set : DINT; (*new V4.13 for ParaBase Counter Set*)
		iCnt_FastStarts_Set : DINT; (*new V4.13 for ParaBase Counter Set*)
		bMsg1995 : BOOL; (*V24*)
		bMsg2000 : BOOL;
		tPB2MM : ParaBase2MM_type; (*USE THIS INTERFACE structure to connect ALL other modules*)
		tPB2AB : MM2AmmBase; (* OWN AlarmBase CONNECTOR as Ammm- Structuretype*)
		tPB2PB : MM2ParaBase_type; (*INTERNAL USE ONLY in PB module! do NOT connect in vvm Selbstgespräche...*) (*OldName: new PV; Cycle: 5;*)
		tSys_Run : HALioDo_Type; (*RUN DigitaOut bit to HAL*) (*OldName: RUN; Cycle: 5;*)
		tSys_Run1 : HALioDo_Type; (*RUN DigitaOut bit to HAL*) (*OldName: RUN; Cycle: 5;*)
		tSys_Run2 : HALioDo_Type; (*RUN DigitaOut bit to HAL*) (*OldName: RUN; Cycle: 5;*)
		tSys_Run3 : HALioDo_Type; (*RUN DigitaOut bit to HAL*) (*OldName: RUN; Cycle: 5;*)
		tSys_Run4 : HALioDo_Type; (*RUN DigitaOut bit to HAL*) (*OldName: RUN; Cycle: 5;*)
		tSys_Run5 : HALioDo_Type; (*RUN DigitaOut bit to HAL*) (*OldName: RUN; Cycle: 5;*)
		tSys_Run6 : HALioDo_Type; (*RUN DigitaOut bit to HAL*) (*OldName: RUN; Cycle: 5;*)
	END_STRUCT;
	MM2VIS_Struct : 	STRUCT
		tPB2VIS : ParaBase2MM_type; (*Uses type of interface to all structure for visu display allso*)
		bDownloadDetected : BOOL := FALSE; (*doppelt?*)
		tModuleState : ARRAY[0..36]OF ModuleInfo_type; (* BUNDELED STATUS INFORMATION of all software modules*)
		bVisVersionClaimsOk : BOOL; (*TRUE=reported VIS version number fits the claimed minimum requirements*)
		tClaimVisVersion : Revision_type;
		bMsg1901 : BOOL;
		bMsg1902 : BOOL;
		bMsg1903 : BOOL;
		bMsg1904 : BOOL;
		bMsg1905 : BOOL;
		bMsg1906 : BOOL;
		bMsg1907 : BOOL;
		bMsg1908 : BOOL;
		bMsg1909 : BOOL;
		bMsg1910 : BOOL;
		bMsg1911 : BOOL;
		bMsg1912 : BOOL;
		bMsg1913 : BOOL;
		bMsg1914 : BOOL;
		bMsg1915 : BOOL;
		bMsg1916 : BOOL;
		bMsg1917 : BOOL;
		bMsg1918 : BOOL;
		bMsg1919 : BOOL;
		bMsg1920 : BOOL;
		bMsg1921 : BOOL;
		bMsg1922 : BOOL;
		bMsg1923 : BOOL;
		bMsg1924 : BOOL;
		bMsg1925 : BOOL;
		bMsg1926 : BOOL;
		bMsg1927 : BOOL;
		bMsg1928 : BOOL;
		bMsg1929 : BOOL;
		bMsg1930 : BOOL;
		bMsg1931 : BOOL;
		bMsg1932 : BOOL;
		bMsg1933 : BOOL;
		bMsg1934 : BOOL;
		bMsg1935 : BOOL;
		bMsg1936 : BOOL;
		bMsg1937 : BOOL;
		bMsg1938 : BOOL;
		bMsg1939 : BOOL;
		bMsg1940 : BOOL;
		bMsg1941 : BOOL;
		bMsg1942 : BOOL;
		bMsg1943 : BOOL;
		bMsg1944 : BOOL;
		bMsg1945 : BOOL;
		bMsg1946 : BOOL;
		bMsg1947 : BOOL;
		bMsg1948 : BOOL;
		bMsg1949 : BOOL;
		bMsg1950 : BOOL;
		bMsg1951 : BOOL;
		bMsg1952 : BOOL;
		bMsg1953 : BOOL;
		bMsg1954 : BOOL;
		bMsg1955 : BOOL;
		bMsg1956 : BOOL;
		bMsg1957 : BOOL;
		bMsg1958 : BOOL;
		bMsg1959 : BOOL;
		bMsg1960 : BOOL;
		bMsg1961 : BOOL;
		bMsg1962 : BOOL;
		bMsg1963 : BOOL;
		bMsg1964 : BOOL;
		bMsg1965 : BOOL;
		bMsg1966 : BOOL;
		bMsg1967 : BOOL;
		bMsg1968 : BOOL;
		bMsg1969 : BOOL;
		bMsg1970 : BOOL;
		bMsg1971 : BOOL;
		bMsg1972 : BOOL;
		bMsg1973 : BOOL;
		bMsg1974 : BOOL;
		bMsg1975 : BOOL;
		bMsg1976 : BOOL;
		bMsg1977 : BOOL;
		bMsg1978 : BOOL;
		bMsg1979 : BOOL;
		bMsg1980 : BOOL;
		bMsg1981 : BOOL;
		bMsg1982 : BOOL;
		bMsg1983 : BOOL;
		bMsg1984 : BOOL;
		bMsg1985 : BOOL;
		bMsg1986 : BOOL;
		bMsg1987 : BOOL;
		bMsg1988 : BOOL;
		bMsg1989 : BOOL;
		bMsg1990 : BOOL;
		bMsg1991 : BOOL;
		iMsg1991 : DINT;
		bMsg1992 : BOOL;
		iMsg1992 : DINT;
		bMsg1993 : BOOL;
		iMsg1993 : DINT;
		bMsg1994 : BOOL;
		iMsg1994 : DINT;
		bMsg1995 : BOOL;
		iMsg1995 : DINT;
		bMsg1996 : BOOL;
		iMsg1996 : DINT;
		bMsg1997 : BOOL;
		iMsg1997 : DINT;
		bMsg1998 : BOOL;
		iMsg1998 : DINT;
		bMsg1999 : BOOL;
		iMsg1999 : DINT;
		bMsg2000 : BOOL;
		iMsg2000 : DINT;
	END_STRUCT;
	VIS2MM_Struct : 	STRUCT
		bParaSaveOnce : BOOL; (*manually initiate a parameter save*)
		iParaSaveOnce_ModuleID : UDINT; (*Module ID code of a single module to save parameter manually. 0 for all modules*)
		bReleasePVI : BOOL; (*restricted!*)
		bRequestPVI : BOOL; (*restricted!*)
		iCnt_OpHours_DataMax : DINT; (* engine operating hours counter (Max Value from VIS DATABASE)*)
		iCnt_OpHours_DataMin : DINT; (* engine operating hours counter (SPARE Min. Value from VIS DATABASE)*)
		iCnt_UnitOpHours_DataMax : DINT; (* unit operating hours counter (Max Value from VIS DATABASE)*)
		iCnt_UnitOpHours_DataMin : DINT; (* unit operating hours counter (SPARE, Min. Value from VIS DATABASE)*)
		iCnt_Starts_DataMax : DINT; (* engine starts counter (Max Value from VIS DATABASE)*)
		iCnt_Starts_DataMin : DINT; (* engine starts counter (SPARE, Minx Value from VIS DATABASE)*)
		iCnt_FastStarts_DataMax : DINT; (* engine starts counter (Max Value from VIS DATABASE)*)
		iCnt_FastStarts_DataMin : DINT; (* engine starts counter (SPARE, Min Value from VIS DATABASE)*)
		iCmd_OpHours_SetCounter : UDINT; (*User command button: 1=set counters, 1+2=3=add to actual counters, 1+8=9=set offset to ignore DB max*)
		iCmd_OpHours_SetCorrMode : UDINT; (*User command button ADD VALUE: 0=set counters, 2=add to actual counters, 8=set offset to ignore DB max*)
		iCnt_OpHours_StoredOffset : DINT; (*ToDo: clarify*)
		iCnt_UnitOpHours_StoredOffset : DINT; (*ToDo: clarify*)
		iCnt_Starts_StoredOffset : DINT; (*ToDo: clarify*)
		iCnt_FastStarts_StoredOffset : DINT; (*ToDo: clarify*)
		tVisVersion : Revision_type;
	END_STRUCT;
END_TYPE
```

### module_PBPara.typ - Para data type. DO NOT CHANGE EXISTING ITEMS!
```iecst
(********************************************************************
 * COPYRIGHT -- INNIO Company
 ********************************************************************
 * Package: ParaBase
 * File: ParaBase.typ
 * Author: zengeres
 * Created: September 14, 2012
 ********************************************************************
 * Para Data type of package ParaBase
  ********************************************************************)

TYPE
	Para_PB : 	STRUCT  (*Para sorting is ok, but add new tags preferably at the end of the para structure*)
		ReplaceMeWithYourParameter : REAL := 1000.0; (*THIS IS JUST A DEMO DATAPOINT! !NOT ON VISU!*)
		iEng_Motortype : INT; (*Para motortype*) (*OldName: new PV; Cycle: 5;*)
		bIgnoreParaSetupOk : BOOL; (*True= allow engine operation without parameter OK*)
		bIgnoreParaSetupOk_AB : BOOL; (*True= allow engine operation without OK from this module*) (*OldName: new PV; Cyclic: 5; ParaID: 11901;*)
		bIgnoreParaSetupOk_AG : BOOL; (*True= allow engine operation without OK from this module*) (*OldName: new PV; Cyclic: 5; ParaID: 11902;*)
		bIgnoreParaSetupOk_CH : BOOL; (*True= allow engine operation without OK from this module*) (*OldName: new PV; Cyclic: 5; ParaID: 11903;*)
		bIgnoreParaSetupOk_CP : BOOL; (*True= allow engine operation without OK from this module*) (*OldName: new PV; Cyclic: 5; ParaID: 11904;*)
		bIgnoreParaSetupOk_CU : BOOL; (*True= allow engine operation without OK from this module*) (*OldName: new PV; Cyclic: 5; ParaID: 11905;*)
		bIgnoreParaSetupOk_EC : BOOL; (*True= allow engine operation without OK from this module*) (*OldName: new PV; Cyclic: 5; ParaID: 11906;*)
		bIgnoreParaSetupOk_EG : BOOL; (*True= allow engine operation without OK from this module*) (*OldName: new PV; Cyclic: 5; ParaID: 11907;*)
		bIgnoreParaSetupOk_EX : BOOL; (*True= allow engine operation without OK from this module*) (*OldName: new PV; Cyclic: 5; ParaID: 11908;*)
		bIgnoreParaSetupOk_GC : BOOL; (*True= allow engine operation without OK from this module*) (*OldName: new PV; Cyclic: 5; ParaID: 11909;*)
		bIgnoreParaSetupOk_GD : BOOL; (*True= allow engine operation without OK from this module*) (*OldName: new PV; Cyclic: 5; ParaID: 11910;*)
		bIgnoreParaSetupOk_GM : BOOL; (*True= allow engine operation without OK from this module*) (*OldName: new PV; Cyclic: 5; ParaID: 11911;*)
		bIgnoreParaSetupOk_GR : BOOL; (*True= allow engine operation without OK from this module*) (*OldName: new PV; Cyclic: 5; ParaID: 11927;*)
		bIgnoreParaSetupOk_GT : BOOL; (*True= allow engine operation without OK from this module*) (*OldName: new PV; Cyclic: 5; ParaID: 11912;*)
		bIgnoreParaSetupOk_HA : BOOL; (*True= allow engine operation without OK from this module*) (*OldName: new PV; Cyclic: 5; ParaID: 11913;*)
		bIgnoreParaSetupOk_HC : BOOL; (*True= allow engine operation without OK from this module*) (*OldName: new PV; Cyclic: 5; ParaID: 11914;*)
		bIgnoreParaSetupOk_IC : BOOL; (*True= allow engine operation without OK from this module*) (*OldName: new PV; Cyclic: 5; ParaID: 11915;*)
		bIgnoreParaSetupOk_IG : BOOL; (*True= allow engine operation without OK from this module*) (*OldName: new PV; Cyclic: 5; ParaID: 11916;*)
		bIgnoreParaSetupOk_KL : BOOL; (*True= allow engine operation without OK from this module*) (*OldName: new PV; Cyclic: 5; ParaID: 11917;*)
		bIgnoreParaSetupOk_KN : BOOL; (*True= allow engine operation without OK from this module*) (*OldName: new PV; Cyclic: 5; ParaID: 11918;*)
		bIgnoreParaSetupOk_MO : BOOL; (*True= allow engine operation without OK from this module*) (*OldName: new PV; Cyclic: 5; ParaID: 11919;*)
		bIgnoreParaSetupOk_OP : BOOL; (*True= allow engine operation without OK from this module*) (*OldName: new PV; Cyclic: 5; ParaID: 11920;*)
		bIgnoreParaSetupOk_PB : BOOL; (*True= allow engine operation without OK from this module*) (*OldName: new PV; Cyclic: 5; ParaID: 11921;*)
		bIgnoreParaSetupOk_SA : BOOL; (*True= allow engine operation without OK from this module*) (*OldName: new PV; Cyclic: 5; ParaID: 11922;*)
		bIgnoreParaSetupOk_SY : BOOL; (*True= allow engine operation without OK from this module*) (*OldName: new PV; Cyclic: 5; ParaID: 11923;*)
		bIgnoreParaSetupOk_TR : BOOL; (*True= allow engine operation without OK from this module*) (*OldName: new PV; Cyclic: 5; ParaID: 11924;*)
		bIgnoreParaSetupOk_VE : BOOL; (*True= allow engine operation without OK from this module*) (*OldName: new PV; Cyclic: 5; ParaID: 11925;*)
		bIgnoreParaSetupOk_VI : BOOL; (*True= allow engine operation without OK from this module*) (*OldName: new PV; Cyclic: 5; ParaID: 11926;*)
		bIgnoreParaSetupOk_28 : BOOL; (*True= allow engine operation without OK from this module*) (*OldName: new PV; Cyclic: 5; ParaID: 11928;*)
		bIgnoreParaSetupOk_TB : BOOL; (*True= allow engine operation without OK from this module*) (*OldName: new PV; Cyclic: 5; ParaID: 11929;*)
		bIgnoreParaSetupOk_OL : BOOL; (*True= allow engine operation without OK from this module*) (*OldName: new PV; Cyclic: 5; ParaID: 11930;*)
		bSaveParaAllowedWithoutSysRun : BOOL; (*True=allow Parameter saving allso if SysRun- bit is missing*) (*OldName: new PV; *)
		bSaveParaAllowedDespiteDownload : BOOL; (*True=allow Parameter saving allso if a DLD- bit is set*) (*OldName: new PV; *)
		bBlockSysRunBit : BOOL; (*True= lock the bBlockSysRun- Signal to FALSE for all modules (for test operation only) !NOT ON VISU!*) (*OldName: new PV; *)
		bDebugShowModuleCount : BOOL; (*true= show module order number, false=ascii module code !NOT ON VISU!*) (*OldName: new PV; *)
		zz_V4_0_ParaVersionEnd : REAL := 4.03; (*! ADD NEW PARAMETER ONLY BELOW THIS LINE ! This is the end of base version parameter and has to stay unchanged. DO NOT CHANGE SORT ORDER of Para!*) (* OldName: new PV; Cycle: 5; *)
		bIgnoreParaSetupOk_EM : BOOL; (*True= allow engine operation without OK from this module*) (*OldName: new PV; Cyclic: 5; ParaID: ;*)
		bIgnoreParaSetupOk_CB : BOOL; (*True= allow engine operation without OK from this module*) (*OldName: new PV; Cyclic: 5; ParaID: ;*)
		iParaBaseExtensionAdress : UDINT; (*prepared; debug only*) (*OldName: new PV; *)
		iParaBaseExtensionCommand : UDINT; (*prepared; debug only*) (*OldName: new PV; *)
	END_STRUCT;
END_TYPE
```

### module_PBPerm.typ - Perm data type. DO NOT CHANGE EXISTING SIZE OR SORTING!
```iecst
TYPE
	PROGRAMMER_INFO_Perm : 	STRUCT
		DO_NOT_CHANGE_PERM : STRING[40] := 'DO NOT CHANGE PERMLENGT OR ELEMENT ORDER'; (* DO NOT ADD OR DELETE ITEMS HERE! *) (*ADD NEW PERM DATAPOINT ONLY BY REPLACING SPARE ENTRIES OF SAME LENGHT!. DO NOT DELETE existing Perm items. Add new file for mayor changes,but avoid changing existing files as long as possible. Every change demands an update of main revision numbering!*)
	END_STRUCT;
	PERM_PB_Struct : 	STRUCT
		iCntDiff_OpHours : DINT; (*********** Parabase Items: start counter 	  ...counter difference*)
		iCntDiff_UnitOpHours : DINT; (*Initial detected counter difference*)
		iCntDiff_Starts : DINT; (*Initial detected  counter difference*)
		iCntDiff_FastStarts : DINT; (*Initial detected  counter difference*)
		iCntUnchanged_OpHours : DINT; (* operating hours counter *)
		iCntUnchanged_UnitOpHours : DINT; (* unit operating hours counter *)
		iCntUnchanged_Starts : DINT; (* start counter *)
		iCntUnchanged_FastStarts : DINT; (* fast start counter *)
		iCnt_Offset_OpHours_DataMax : DINT; (*V4.13   holds possible offset to surpress warning*)
		iCnt_Offset_UnitOpHours_DataMax : DINT; (*V4.13   holds possible offset to surpress warning*)
		iCnt_Offset_Starts_DataMax : DINT; (*V4.13   holds possible offset to surpress warning*)
		iCnt_Offset_FastStarts_DataMax : DINT; (*V4.13   holds possible offset to surpress warning ?*)
		iCmd_OpHours_SetCounter : UDINT; (*V4.13   holds commands and execution date to surpress warning ?*)
		iCmd_ReduceStoredOffsets : UDINT; (*V4.13   holds commands and flags to surpress warning ?*)
		tCommand_Execution_Time : RTCtime_typ; (*V4.13   holds execution time to surpress warning ?*)
		tDetectedEvent_Time : RTCtime_typ; (*V4.13   suspected time of counter failure *)
		tSpare_Time : RTCtime_typ; (*V4.13   holds room for future*)
		iCnt_OpHours : DINT; (* operating hours counter *) (*OldName:betrieb_h;Cycle:2;*)
		iCnt_UnitOpHours : DINT; (* unit operating hours counter *)
		iCnt_Starts : DINT; (*********** Backup Opstate: start counter *) (*OldName:start_z;Cycle:2;*)
		iCnt_FastStarts : DINT; (* fast start counter *)
		rPB_PermValue01 : REAL; (********** spare permanent value - replace with new vars of same lenght, when needed*)
		rPB_PermValue02 : REAL; (*spare permanent value - replace with new vars of same lenght, when needed*)
		rPB_PermValue03 : REAL; (*spare permanent value - replace with new vars of same lenght, when needed*)
		rPB_PermValue04 : REAL; (*spare permanent value - replace with new vars of same lenght, when needed*)
		rPB_PermValue05 : REAL; (*spare permanent value - replace with new vars of same lenght, when needed*)
		rPB_PermValue06 : REAL; (*spare permanent value - replace with new vars of same lenght, when needed*)
		rPB_PermValue07 : REAL; (*spare permanent value - replace with new vars of same lenght, when needed*)
		rPB_PermValue08 : REAL; (*spare permanent value - replace with new vars of same lenght, when needed*)
		rPB_PermValue09 : REAL; (*spare permanent value - replace with new vars of same lenght, when needed*)
		rPB_PermValue10 : REAL; (*spare permanent value - replace with new vars of same lenght, when needed*)
		rPB_PermValue11 : REAL; (*spare permanent value - replace with new vars of same lenght, when needed*)
		rPB_PermValue12 : REAL; (*spare permanent value - replace with new vars of same lenght, when needed*)
		rPB_PermValue13 : REAL; (*spare permanent value - replace with new vars of same lenght, when needed*)
		rPB_PermValue14 : REAL; (*spare permanent value - replace with new vars of same lenght, when needed*)
		rPB_PermValue15 : REAL; (*spare permanent value - replace with new vars of same lenght, when needed*)
		rPB_PermValue16 : REAL; (*spare permanent value - replace with new vars of same lenght, when needed*)
		rPB_PermValue17 : REAL; (*spare permanent value - replace with new vars of same lenght, when needed*)
		rPB_PermValue18 : REAL; (*spare permanent value - replace with new vars of same lenght, when needed*)
		rPB_PermValue19 : REAL; (*spare permanent value - replace with new vars of same lenght, when needed*)
		rPB_PermValue20 : REAL; (*spare permanent value - replace with new vars of same lenght, when needed*)
		rPB_PermValue21 : REAL; (*spare permanent value - replace with new vars of same lenght, when needed*)
		rPB_PermValue22 : REAL; (*spare permanent value - replace with new vars of same lenght, when needed*)
		rPB_PermValue23 : REAL; (*spare permanent value - replace with new vars of same lenght, when needed*)
		rPB_PermValue24 : REAL; (*spare permanent value - replace with new vars of same lenght, when needed*)
		rPB_PermValue25 : REAL; (*spare permanent value - replace with new vars of same lenght, when needed*)
		rPB_PermValue26 : REAL; (*spare permanent value - replace with new vars of same lenght, when needed*)
		rPB_PermValue27 : REAL; (*spare permanent value - replace with new vars of same lenght, when needed*)
		rPB_PermValue28 : REAL; (*spare permanent value - replace with new vars of same lenght, when needed*)
		rPB_PermValue29 : REAL; (*spare permanent value - replace with new vars of same lenght, when needed*)
		rPB_PermValue30 : REAL; (*spare permanent value - replace with new vars of same lenght, when needed*)
		rPB_PermValue31 : REAL; (*spare permanent value - replace with new vars of same lenght, when needed*)
		rPB_PermValue32 : REAL; (*spare permanent value - replace with new vars of same lenght, when needed*)
		rPB_PermValue33 : REAL; (*spare permanent value - replace with new vars of same lenght, when needed*)
		rPB_PermValue34 : REAL; (*spare permanent value - replace with new vars of same lenght, when needed*)
		rPB_PermValue35 : REAL; (*spare permanent value - replace with new vars of same lenght, when needed*)
		rPB_PermValue36 : REAL; (*spare permanent value - replace with new vars of same lenght, when needed*)
		rPB_PermValue37 : REAL; (*spare permanent value - replace with new vars of same lenght, when needed*)
		rPB_PermValue38 : REAL; (*spare permanent value - replace with new vars of same lenght, when needed*)
		rPB_PermValue39 : REAL; (*spare permanent value - replace with new vars of same lenght, when needed*)
		rPB_PermValue40 : REAL; (*spare permanent value - replace with new vars of same lenght, when needed*)
		rPB_PermValue41 : REAL; (*spare permanent value - replace with new vars of same lenght, when needed*)
		rPB_PermValue42 : REAL; (*spare permanent value - replace with new vars of same lenght, when needed*)
		rPB_PermValue43 : REAL; (*spare permanent value - replace with new vars of same lenght, when needed*)
		rPB_PermValue44 : REAL; (*spare permanent value - replace with new vars of same lenght, when needed*)
		rPB_PermValue45 : REAL; (*spare permanent value - replace with new vars of same lenght, when needed*)
		rPB_PermValue46 : REAL; (*spare permanent value - replace with new vars of same lenght, when needed*)
		rPB_PermValue47 : REAL; (*spare permanent value - replace with new vars of same lenght, when needed*)
		rPB_PermValue48 : REAL; (*spare permanent value - replace with new vars of same lenght, when needed*)
		rPB_PermValue49 : REAL; (*spare permanent value - replace with new vars of same lenght, when needed*)
		rPB_PermValue50 : REAL; (*spare permanent value - replace with new vars of same lenght, when needed*)
		iCnt_IslandHours : DINT; (* spare preparation only! island operating hours counter*)
		iCnt_NetPHours : DINT; (* spare preparation only! net parallel operating hours counter*)
		iCnt_DemHours : DINT; (* spare preparation only! demanded hours counter*)
		iIdx_OMSS : DINT; (*spare preparation only!  operation mode selector switch *)
		iIdx_RSS : DINT; (*spare preparation only!  remote selector switch *)
	END_STRUCT;
END_TYPE
```

### ParaBase.var - Package variables
```iecst
(********************************************************************
 * COPYRIGHT -- INNIO Company
 ********************************************************************
 * Package: ParaBase
 * File: ParaBase.var
 * Author: zengeres
 * Created: September 17, 2012
 ********************************************************************
 * Variables of package ParaBase
 ********************************************************************)
VAR
	IN_PB : IN_PB_Struct;
	OUT_PB : OUT_PB_Struct;
	MM2VIS : MM2VIS_Struct;
	VIS2MM : VIS2MM_Struct;
	Para : Para_PB;
	ParaFactoryDefault : Para_PB := (0);
	pm : Para_PB;
	bOMSS_Stop : BOOL; (*engine operation mode selection*)
	bOMSS_Man : BOOL; (*engine operation mode selection*)
	bOMSS_Aut : BOOL; (*engine operation mode selection*)
	bOMSS_Test : BOOL; (*engine operation mode selection*)
	bOMSS_Scav : BOOL; (*engine operation mode selection*)
	bOMSS_MAT : BOOL; (*engine operation mode selection*)
	bForceModuleMandatory_VE : BOOL;
	bForceModuleMandatory_HC : BOOL;
	bForceModuleMandatory_EX : BOOL;
	bForceModuleMandatory_TR : BOOL;
	bForceModuleMandatory_GC : BOOL;
	bForceModuleMandatory_CU : BOOL;
	bForceModuleMandatory_MO : BOOL;
	bForceModuleMandatory_IC : BOOL;
	bForceModuleMandatory_IG : BOOL;
	bForceModuleMandatory_GR : BOOL;
	bForceModuleMandatory_SY : BOOL;
	bForceModuleMandatory_CP : BOOL;
	bForceModuleMandatory_EC : BOOL;
	bForceModuleMandatory_EG : BOOL;
	bForceModuleMandatory_EM : BOOL;
	bForceModuleMandatory_KN : BOOL;
	bForceModuleMandatory_GM : BOOL;
	bForceModuleMandatory_GT : BOOL;
	bForceModuleMandatory_AG : BOOL;
	bForceModuleMandatory_OP : BOOL;
	bForceModuleMandatory_SA : BOOL;
	bForceModuleMandatory_KL : BOOL;
	bForceModuleMandatory_GD : BOOL;
	bForceModuleMandatory_CH : BOOL;
	bForceModuleMandatory_HA : BOOL;
	bForceModuleMandatory_AB : BOOL;
	bForceModuleMandatory_VI : BOOL;
	bForceModuleMandatory_CB : BOOL;
	bForceModuleMandatory_PB : BOOL; (*(MYSELF)*)
	bParaReadBackRelease : BOOL; (*has to be true to allow parameter restore*)
	iTestMissingParaModule : DINT; (*prepared*)
	iNoOfFirstParaMissing : DINT; (*iNoOfFirstParaMissing*)
	iNoOfFirstParaWarnings : DINT;
	iNoOfFirstPermMissing : DINT; (*new V4.06*)
	iIDOfFirstPermMissing : DINT; (*new V4.06*)
	szFirstPermMissing : STRING[2]; (*new V4.06*)
	bPermMissingError : BOOL; (*new V4.06*)
	iDebugFirstMissing_SysRun : DINT;
	iDebugFirstMissing_DLD : DINT; (*prepared*)
	bNoInitDetected : BOOL := FALSE; (*allways true, except 1cycle on init up*)
	bErr_PermStore : ARRAY[0..31] OF BOOL; (*V4.13   Alarmbits for unplausible Perm values*)
	Perm : PERM_PB_Struct; (*Values permanetly stored in Flash Datamodule*)
	pm1 : PERM_PB_Struct; (*Flash Datamodule*)
END_VAR
```

### Program Logical/ParaBase/ParXX_TEMPLATE (IEC, version 4.00.0) - + parameter storage and modulstate communication

- perm_par.st (not readable text: treated as protected, skipped)

### Program Logical/ParaBase/setting_PB (IEC, version 4.03.0) - + cofiguration for basic system checks

#### setting_PBInit.st
```iecst
(*******************************************************************************
settings			meta module settings

This code is confidential and proprietary to the INNIO Company.
It may not be used in any form, or reproduced in any manner,
without the express written permission of the INNIO Company.
Copyright, INNIO Company, 2019

Customized modifications: -
------------------------

History:
-------
V0.1	17.09.2012	Zengerer	new
V4.03	30.10.2015	Zengerer	bForceModuleMandatory_KN := TRUE

Instructions for use:
--------------------
cofiguration storage for some basic system checks

Outstandings:
------------

(*******************************************************************************)
PROGRAM _INIT
												(* old_var:		comment:												unit:	def:	min:	max:	read:	write:	*)
	Para.iEng_Motortype;		(*	:=	412;	(* x			Para engine motortype									n/a		920		208		920		10		50		*)

	(* Configure optional Factory Default Values here, if no datamodule exists on a new/empti controller *)
	ParaFactoryDefault.bSaveParaAllowedDespiteDownload :=	TRUE;
	ParaFactoryDefault.bIgnoreParaSetupOk_TR := 			TRUE;
	ParaFactoryDefault.ReplaceMeWithYourParameter :=		54321;	(*Demo value, no function*)

	(* Configure MANDATORY Metamodules here HARDCODED *)
	bForceModuleMandatory_AB := TRUE;
	bForceModuleMandatory_AG;
	bForceModuleMandatory_CH;
	bForceModuleMandatory_CP;
	bForceModuleMandatory_CU;
	bForceModuleMandatory_EC := TRUE;
	bForceModuleMandatory_EG;
	bForceModuleMandatory_EM;				(*Exhaust Monitoring, new*)
	bForceModuleMandatory_EX;
	bForceModuleMandatory_GC;
	bForceModuleMandatory_GD;
	bForceModuleMandatory_GM;
	bForceModuleMandatory_GR; (*prepared*)
	bForceModuleMandatory_GT;
	bForceModuleMandatory_HA := TRUE;
	bForceModuleMandatory_HC;
	bForceModuleMandatory_IC;
	bForceModuleMandatory_IG;
	bForceModuleMandatory_KL;
	bForceModuleMandatory_KN := TRUE;
	bForceModuleMandatory_MO;
	bForceModuleMandatory_OP := TRUE;
	bForceModuleMandatory_PB := TRUE;
	bForceModuleMandatory_SA;
	bForceModuleMandatory_SY;
	bForceModuleMandatory_TR;
	bForceModuleMandatory_VE;
	bForceModuleMandatory_VI;

	//CANCELLED: AUSLESEN DIESER INFO AUS MODUL- METAINFO FILE?

	IN_PB.tAlarmB2PB.bResetTrip; 	(*Fehlt noch: Amm- Anbindung der ParaBase- eigenen Alarme*)
	OUT_PB.tPB2AB.bGnlWarning;		(*Fehlt noch: Amm- Anbindung der ParaBase- eigenen Alarme*)

END_PROGRAM
```

### Program Logical/ParaBase/general_PB (IEC, version 4.02.0) - + general functions

- general_PBCyclic.st (not readable text: treated as protected, skipped)

#### general_PB.var
```iecst
VAR
	xEngType : EngType;
	xOpMode : OpMode;
END_VAR
```

### Program Logical/ParaBase/ParPB (IEC, version 4.06.0) - + parameter handling

- perm_par.st (not readable text: treated as protected, skipped)

#### perm_par.var
```iecst
VAR
	tParaIntern : ParaHandler_typ; (*Connector type to perm_par*)
	tMM2ParaBase_ReadBack : MM2ParaBase_type; (*INTERNAL! V4.06 new readback structure for information from previous tasks*)
	bWriteDataObj : BOOL; (* TRUE=write data object module *)
	bDataObjLenErr : BOOL; (*Error occured in permem: data module size missmatch*)
	bCreateDataObj : BOOL; (* TRUE=create new data object *)
	bWriteOnce : BOOL; (* write permanent memory once *)
	DatObjCreate_01 : DatObjCreate; (* data object create *)
	DatObjInfoBak_02 : DatObjInfo; (* data object info *)
	DatObjDelete_01 : DatObjDelete; (* data object delete *)
	DatObjRead_01 : DatObjRead; (* data object read *)
	DatObjRead_02 : DatObjRead; (* manual initiated data object read *)
	DatObjWrite_01 : DatObjWrite; (* data object write *)
	DatObjDelete_02 : DatObjDelete; (* data object delete *)
	DatObjDelete_11 : DatObjDelete; (*Delete Backup File*)
	DatObjInfo_01 : DatObjInfo; (* data object info *)
	DatObjInfo_02 : DatObjInfo; (* data object info *)
	szModuleName : STRING[35]; (* module name of object *)
	szModuleNameBackup : STRING[35]; (* module name of posiibly created backup object *)
	DatObjCopy_01 : DatObjCopy;
	bCopyDataObj : BOOL;
	TON_WarnDelay : TON;
	TON_WritePMEM : TON; (* delay write permanent memory *)
	ulPMPointer : UDINT; (* adress of actual checksum value *)
	ulChecksum : UDINT; (* parameter checksum value *)
	pm_len : UDINT; (* permanent value lenght *)
	ulChecksumOld : UDINT; (* last vlaue of parameter checksum *)
	ulChkValue : UDINT; (* actual value of parameter pointer *)
	pm_id : UDINT; (* permanent value identifier *)
	pm_p : UDINT; (* permanent value pointer *)
	DatObjInfo_META : DatObjInfo;
	DatObjRead_META : DatObjRead;
	szMetaDataRaw : STRING[2000];
	szMetaData : ARRAY[0..4] OF STRING[35];
	szMetaDataVis : ARRAY[0..3] OF STRING[35];
	ssIndex : INT;
	ssCount : INT;
	ucMetaDataRaw : ARRAY[0..2000] OF USINT;
	ssCount2 : INT;
	szMetaDataFile : STRING[10];
	szText1 : STRING[20];
	pv_adr_IN_XX_tPB2MM : UDINT;
	pv_lng : UDINT;
	pv_lng_IN_XX_tPB2MM : UDINT;
	pv_lng_OUT_XX_tPB2MM : UDINT;
	szText2 : STRING[20];
	pv_adr_OUT_XX_tXX2PB : UDINT;
END_VAR
VAR CONSTANT
	ERR_NOERROR : UINT := 0;
END_VAR
VAR
	usPMWriteCnt : UINT;
	pm_Error : UDINT; (* permanent value error *) (* Deleted: pm : ParaMem_typ; permanent memory tags mathias, 22.8.11*)
	fun_Error : UDINT := 0; (*state > 0 = function error*)
	xLocalParaCheck : ParaCheckFUB; (*local function instance to check parameter values*)
	TON_ParaSetupOk : TON;
	bParaCheckSystemOk : BOOL;
	iDebug_ParaOkChecked : UDINT;
	bRestoreBackupDataObj : BOOL := FALSE;
	bRestoreDataObjContent : BOOL := FALSE;
	pm_id_backup : UDINT;
	pm_p_Backup : UDINT;
	DatObjCopy_02 : DatObjCopy;
	bDeleteBackupDataObj : BOOL := FALSE; (*Command to delete backup data module file on purpose*)
	bDebugPara : ARRAY[0..5] OF BOOL;
	ssIndex2 : INT;
	ssIndex3 : INT;
	ssIndex4 : INT;
	ssIndexVis : INT;
	szText : STRING[40];
	pv_adr_Para : UDINT;
	szParaSnippet : ARRAY[0..5] OF STRING[150];
	szParaIndex : STRING[10];
	slValue : DINT;
	iModuleDLD_ResetCount : INT;
	bDownloadDetected : BOOL;
	bFlagParaStructCopyWorking : BOOL; (*true, if cyclic para copying is active, 1 false cycle at every copy *)
	bStoreInitParaInDataObj : BOOL := FALSE;
	bTestflag : BOOL;
	bReadOutMETA_Once : BOOL;
	tParaCheck_iPvAdress : ARRAY[0..5] OF UDINT;
	tParaCheck_iPvLengt : ARRAY[0..5] OF UDINT;
	tParaCheck_rPvValue : ARRAY[0..5] OF REAL;
	tParaCheck_rRangeMIN : ARRAY[0..5] OF REAL;
	tParaCheck_rRangeMAX : ARRAY[0..5] OF REAL;
	tParaCheck_szPvName : ARRAY[0..5] OF STRING[35];
	ssFormatDetected : INT;
	szMetaDataPart : STRING[150];
	szFullTaskName : STRING[35];
	szFullMetaModuleName : STRING[35];
	debugLen : INT;
	debugSize : INT := 0;
	strcat_adr1 : UDINT;
	strcat_adr2 : UDINT;
	ssIndexTN : INT;
	bAlternate : BOOL;
	n : INT;
	iAlternateChecksum : DINT;
	iAlternateChecksumOld : DINT;
	ulDebugChkValue : ARRAY[0..999] OF UDINT;
	Adr1 : UDINT;
	Adr2 : UDINT;
	usPMWriteCntStepsize : UINT := 1; (*different step sizes to help debug*)
	usPMWriteCntXOR : UINT;
	usPMWriteCntAltSum : UINT;
	ulAdrPM : UDINT;
	usChkValuePM : USINT;
	ulAdrPara : UDINT;
	ulPara_len : UDINT;
	usChkValuePara : USINT;
	iDebugCountPMDifferences : DINT := 0;
	bEngineRunDetected : BOOL; (*detection status bit autocommand 100 /101  for engine run state*)
	ucMetaDataDebugInfoLine : ARRAY[0..24] OF STRING[80];
	ssIndexMand : INT := 0;
	szMetaDataMand : STRING[35];
	iMyErrorInfo_Autoreset : DINT; (*internal autoreset counter*)
	ssIndex_Version : INT; (*internal*)
	ssIndex_BU : INT; (*internal*)
	ssIndex_BU2 : INT; (*internal*)
END_VAR
```

### Program Logical/ParaBase/ParaMaster (IEC, version 4.03.0) - + communication master to all metamodules

- ParaMasterCyclic.st (not readable text: treated as protected, skipped)

- ParaMasterInit.st (not readable text: treated as protected, skipped)

#### ParaMaster.var
```iecst
VAR
	bParaSetupOk : BOOL;
	TON_ParaSetupOk : TON;
	sRefTestMissingParaModule : REFERENCE TO STRING[2];
	sTestMissingParaModule : STRING[2];
	iTest : UDINT;
	cnt : INT;
	iCountParaSetupOk : INT; (*Debug counter for modules stated OK*)
	iCountParaSetupFailed : INT; (*Debug counter for modules missing AND NOT DISABELED PER PARAMETER*)
	iCountParaWarnings : INT; (*Debug counter for modules with parameter warnings*)
	iCountParaMissing : INT;
	iDebugCount_SysRunOk : INT;
	TON_SysRun : TON;
	iDebugCount_DLD : INT;
	bBlockDownloadDetect_DEBUG : BOOL := FALSE; (*for debugging only!*)
	bDEBUG_SetSys_Run : BOOL := FALSE;
	bDebugSysRunOk : ARRAY[0..36] OF BOOL; (*nur ein praktisches Array für einfache Watch Darstellung*)
	iDebug_Prog_Vers_Simple : ARRAY[0..36] OF UDINT; (*Debug Modulversion mit bMySysRun verknüpft*)
	bBlinkDebugActive : BOOL; (*intern*)
END_VAR
VAR CONSTANT
	eActivateDebugBlink : DINT := 7; (*lokal command value: toggle DebugBlink*)
	eDeactivateAutoCommands : DINT := 100; (*lokal command value: bSendAutoCommands off*)
	eActivateAutoCommands : DINT := 101; (*lokal command value: bSendAutoCommands on*)
END_VAR
VAR
	bSendAutoCommands : BOOL := FALSE; (*Debug Value: starts cyclic command send with engine on/off info*)
	TON_WritePMEM : TON;
	bEngineRunDetected : BOOL; (*here DEBUG INFORMATION  only*)
	TON_ResetExt : TON;
	iDebugCount_Perm : INT := 0; (*V4.06*)
	iDebugFirstMissing_Perm : UDINT := 0; (*V4.06*)
	bOptShowNegPermStatus : BOOL := TRUE; (*V4.06 prepared*)
END_VAR
```

### Program Logical/ParaBase/VisVersion (IEC, version 4.04.2) - + Collect the necessary version numbers for the VIS

- VisVersionCyclic.st (not readable text: treated as protected, skipped)

- VisVersionInit.st (not readable text: treated as protected, skipped)

#### VisVersion.var - Lokale Variablen
```iecst
(********************************************************************
 * COPYRIGHT -- INNIO Company
 ********************************************************************
 * Programm: VisVersion
 * Datei: VisVersion.var
 * Autor: zengeres
 * Erstellt: 9. April 2014
 ********************************************************************
 * Lokale Variablen des Programms VisVersion
 ********************************************************************)
VAR
	cnt : DINT;
	iCountVisVersionStatements : DINT;
	iCountWrongVisVersionClaims : DINT;
	bErrWrongVisVersionClaims : BOOL;
	bDoNoVisVersionClaimsCheck : BOOL := FALSE; (*Debug flag to surpress version check message*)
	bDoNoExactMajorVisVersionCheck : BOOL := FALSE; (*Debug flag to surpress exact mayor version check, TRUE is a >= check only*)
	iModuleIDClaimingWrongVisVersion : UDINT;
END_VAR
```

### Program Logical/ParaBase/CheckMap (ANSIC) - + Check for unresolved PV2PV mappings

#### CheckMap.c - Implementation code
```c
/********************************************************************
 * COPYRIGHT --
 ********************************************************************
 * Program: CheckMap
 * File: CheckMap.c
 * Author: havlovect
 * Created: September 27, 2011
 ********************************************************************
 * Programm zum Auslesen von inaktiven PV-PV Rangierungen
 * Zum Starten muss man die "state" Variable auf 1 setzen
 * Nach einem erfolgreichen Durchlauf ist dann "state" auf 1000
 * und in der Tabelle "Table" sind "table_index" Eintraege mit inaktiven
 * PV-PV Rangierungen.
 * Im Fehlerfall hat "state" den Wert 999, und "errState" gibt den
 * Schritt in der State-Machine an, in dem der Fehler auftrat
 ********************************************************************/

#include <bur/plctypes.h>

#ifdef _DEFAULT_INCLUDES
	#include <AsDefault.h>
#endif

#include <string.h>

#define INIT_MAPPING_S            1
#define NEXT_MAPPING_S           10
#define INIT_LINK_S				 15
#define LINK_S					 20
#define ERROR_S					999
#define RETRY_MAPPING_S			500
#define FINISHED_S			   1000

static void clear_table()
/* Loeschen der Tabelle mit den Resultaten */
{
	table_index = 0;
	memset (&Table, 0, sizeof(Table));
}

static void insert_entry(char * sourceName,
						 USINT  sourceFlags,
						 char * sinkName,
	                     USINT  sinkFlags)
	/* Eintrag eines Resultats in die Tabelle
	   Hier waeren eventuell noch weitere Filterungen moeglich,
	   z.B. nur Rangierungen eintragen, deren Ziel in einem bestimmten
	   AppModul liegen.
	*/
{
	if (table_index <= MAX_TABLE)
	{
		strncpy(Table[table_index].sourceName, sourceName, sizeof(Table[0].sourceName));
		strncpy(Table[table_index].sinkName,   sinkName,   sizeof(Table[0].sinkName));
		Table[table_index].sourceFlags = sourceFlags;
		Table[table_index].sinkFlags   = sinkFlags;

		table_index++;
	}
}

void _INIT CheckMapINIT(void)
{
	state = 1;		/* Start automatisch mit PLC Hochlauf */
	AsArLogGetInfo_01.enable = 1;
	AsArLogGetInfo_01.pName = arlogBASE_USER_LOG_IDENT;
	AsArLogGetInfo(&AsArLogGetInfo_01);
}

void _CYCLIC CheckMapCYCLIC(void)
{
	if (active)
		cycleCount++;

	switch (state) {
		case INIT_MAPPING_S:
		/* Einstieg in die State-Machine, Initialisierung des Loops ueber AsIOFListDP */

			cycleCount = 0;
			active = 1;
			clear_table();
			/* Wir interessieren uns nur fuer PV-PV Rangierungen, die nicht aktiv sind
			   (siehe Dokumentation des FUBs) */
			List.flagsMask      = 0x38;
			List.flagsValue     = 0x08;

			List.enable         = 1;
			List.pLastDatapoint = 0;
			state = NEXT_MAPPING_S;
			/* FALLTHROUGH */
		case NEXT_MAPPING_S:
		/* Aufruf von AsIOFListDP */

			AsIOFListDP(&List);
			if (List.status == ERR_FUB_BUSY)
			{
				/* weiter aufrufen */
				break;
			}
			/* FUB ist fertig geworden -> Auswertung */

			if (List.status == asioERR_NOSUCH_DP)
			{
				/* Datenpunkt inzwischen verschwunden -> nochmals von vorne beginnen */
				state = RETRY_MAPPING_S;
				break;
			}

			/* Behandlung anderer Fehler */
			if (List.status != ERR_OK)
			{
				errState = NEXT_MAPPING_S;
				active = 0;
				state = ERROR_S;
				break;
			}

			/* FUB ist erfolgreich fertig geworden */

			if (List.pDatapoint == 0)
			{
				/* Kein weiterer Eintrag mehr gefunden -> Fertig */
				active = 0;
				state = FINISHED_S;
				break;
			}

			/* Wir haben einen passenden Datenpunkt gefunden */

			/* Fuer naechsten Durchlauf pLastDatapoint weitersetzen */
			List.pLastDatapoint = List.pDatapoint;

			state = INIT_LINK_S;
			/* FALLTHROUGH */
		case INIT_LINK_S:
		/*	die betroffenen PVs auswerten: Initialisierung fuer AsIOPVInfo */

			str[0][0] = 0;
			str[1][0] = 0;
			lflags[0] = 0;
			lflags[1] = 0;

			Info.enable = 1;
			Info.pDatapoint = List.pDatapoint;

			/* Mit Signalquelle (index 0) starten */
			Info.index = 0;
			state = LINK_S;
			/* FALLTHROUGH */
		case LINK_S:
		/* Aufruf von AsIOPVInfo */

			AsIOPVInfo(&Info);
			if (Info.status == ERR_FUB_BUSY)
			{
				/* weiter aufrufen */
				break;
			}
			/* FUB ist fertig geworden -> Auswertung */

			if (Info.status == asioERR_NOSUCH_DP)
			{
				state = RETRY_MAPPING_S;
				break;
			}

			/* Behandlung anderer Fehler */
			if (Info.status != ERR_OK)
			{
				errState = LINK_S;
				active = 0;
				state = ERROR_S;
				break;
			}

			/* FUB ist erfolgreich fertig geworden */

			if (Info.pPvName)
				strncpy(str[Info.index], (char *)Info.pPvName, sizeof(str[Info.index]));
			lflags[Info.index] = Info.flags;

			if (Info.index == 0)
			{
				/* Wir haben die Signalquelle ausgelesen und wollen
				   jetzt die erste Senke auslesen:
				   index auf 1 setzen, aber im gleichen State bleiben */
				Info.index = 1;
				break;
			}

			/* Wir haben jetzt auch die erste Senke ausgelesen,
			   und da es bei PV-PV Rangierungen nur eine Senke gibt, sind
               wir jetzt fertig */

			/* Merken der Rangierung */
			insert_entry(str[0], lflags[0], str[1], lflags[1]);

			/* und weiter im Loop mit AsIOFListDP */
			state = NEXT_MAPPING_S;
			break;
		case RETRY_MAPPING_S:
		/*  Falls waehrend der Abarbeitung durch Deinstall von Mapping Modulen
			der letzte/aktuelle Datenpunkt nicht gefunden wurde fangen wir nochmals von vorne an
	     */
			retryCount++;
			state = INIT_MAPPING_S;
			break;
		case FINISHED_S:
		/*  Logger Eintrag der inaktiven Mappings */
			strcpy(logErrorStringPV, "There are ");
			strcpy(hilfstr2, " unresolved PV2PV mappings. For details see: ParaBase::Checkmap.Table");
			itoa(table_index,(UDINT)hilfstr3);
			strcat(logErrorStringPV, hilfstr3);
			strcat(logErrorStringPV, hilfstr2);

         	AsArLogWrite_01.enable = 1;
			AsArLogWrite_01.ident = AsArLogGetInfo_01.ident;
			AsArLogWrite_01.logLevel = arlogLEVEL_WARNING;
			AsArLogWrite_01.errornr = 52200;
			AsArLogWrite_01.asciiString = (UDINT)(&logErrorStringPV);
			AsArLogWrite(&AsArLogWrite_01);
			if (AsArLogWrite_01.status != 0)
				state = 0;
			break;
		default:
			break;
	}
}
```

#### CheckMap.typ - Local data types
```iecst
(********************************************************************
 * COPYRIGHT --
 ********************************************************************
 * Program: CheckMap
 * File: CheckMap.typ
 * Author: havlovect
 * Created: September 27, 2011
 ********************************************************************
 * Local data types of program CheckMap
 ********************************************************************)

TYPE
	TableEntry : 	STRUCT
		sourceName : STRING[255]; (*Name der Quell PV*)
		sourceFlags : USINT;
		sinkName : STRING[255]; (*Name der Ziel PV*)
		sinkFlags : USINT;
	END_STRUCT;
END_TYPE
```

#### CheckMap.var - Local variables
```iecst
(********************************************************************
 * COPYRIGHT --
 ********************************************************************
 * Program: CheckMap
 * File: CheckMap.var
 * Author: havlovect
 * Created: September 27, 2011
 ********************************************************************
 * Local variables of program CheckMap
 ********************************************************************)
VAR
	state : UDINT; (*State-Machine Steuerung*)
END_VAR
VAR CONSTANT
	MAX_TABLE : UDINT := 100;
END_VAR
VAR
	retryCount : UDINT;
	Info : AsIOPVInfo; (*FUB Instanz*)
	List : AsIOFListDP; (*FUB Instanz*)
	errState : UDINT; (*Schritt der Statemachine, in der ein Fehler auftrat*)
	cycleCount : UDINT; (*Anzahl der Zyklen bei fuer einen vollstaendigen Durchlauf*)
	str : ARRAY[0..1] OF STRING[256]; (*Hilfsvariable*)
	lflags : ARRAY[0..1] OF USINT; (*Hilfsvariable*)
	active : BOOL; (*State-Machine ist in Abarbeitung*)
	Table : ARRAY[0..MAX_TABLE] OF TableEntry; (*Ergebnistabelle*)
	table_index : UDINT; (*Anzahl Tabelleneintraege*)
	AsArLogWrite_01 : AsArLogWrite := (0);
	AsArLogGetInfo_01 : AsArLogGetInfo := (0);
	logErrorStringPV : STRING[256];
	hilfstr2 : STRING[200];
	hilfstr3 : STRING[200];
END_VAR
```

### Program Logical/ParaBase/PermCntCheck (IEC, version 4.13.1) - + Check counter integrity

- PermCntCheckCyclic.st (not readable text: treated as protected, skipped)

- PermCntCheckInit.st (not readable text: treated as protected, skipped)

#### PermCntCheck.var
```iecst
VAR
	bTrig_Cnt_Set : BOOL; (*internal*)
	TON_Trig_Cnt_Set : TON;
	usStatus_gettime : UINT;
	tGetTime : RTCtime_typ; (*clock time*)
	iGetTime : UDINT; (*date/clock time converted*)
	cnt : USINT := 0;
END_VAR
VAR CONSTANT
	iConst_TimeSimpleYear : UDINT := 2000; (*2000 or 2020 as constant to reduction ofcalendaryear  to 2 or 1 digits, to reduce integer value*)
END_VAR
VAR
	iCnt_Tolerance : DINT := 1;
	bOpt_AllwaysSetAllCnt : BOOL := FALSE; (*FALSE only corrects lower counters, that have detected errors (those that are lower than database values).*)
END_VAR
```

### Program Logical/ParaBase/MsgPB (IEC, version 4.13.0) - + Alarms generation

- MsgPBCyclic.st (not readable text: treated as protected, skipped)

- MsgPBInit.st (not readable text: treated as protected, skipped)

#### MsgPB.var
```iecst
VAR
	iAdrAmmBase2MM : UDINT;
	iAdrMM2AmmBase : UDINT;
	xMsg1901 : Msg; (*FuB*)
	xMsg19 : ARRAY[0..99] OF Msg; (*Array of FuBs*)
	xMsg2000 : Msg;
	bBlockMsg19 : ARRAY[0..99] OF BOOL;
	cnt : UDINT;
	bDisableSysWarnings : BOOL; (*True disabeles para system warnings (if engine is already running)*)
	xOpMode : OpMode;
	iModuleCnt : UDINT;
	bParaMessageError : BOOL;
	iMsg19_Size : UDINT; (*internal array range check*)
	iModuleState_Size : UDINT;
	bBlockRebootMessages : BOOL;
	TON_Reboot : TON := (0);
	bBlock_ForwardingMsg1995 : BOOL := TRUE; (*debug *)
	bBlock1995 : BOOL := FALSE; (*debug only*)
	bBlock1996 : BOOL := FALSE; (*debug only*)
	bOpt_AutoReset_1996 : BOOL := TRUE; (*W1996 Counter value error Allways TRUE according to CDR 07.11.23*)
END_VAR
```

### Program Logical/ParaBase/PermPB (IEC, version 4.13.0) - + Permanent variable storage PB

- PermPBCyclic.st (not readable text: treated as protected, skipped)

- PermPBInit.st (not readable text: treated as protected, skipped)

#### PermPB.var
```iecst
VAR
	tParaIntern : ParaHandler_typ; (*Connector type to perm_par*)
	bWriteDataObj : BOOL; (* TRUE=write data object module *)
	bDataObjLenErr : BOOL; (*Error occured in permem: data module size missmatch*)
	bCreateDataObj : BOOL; (* TRUE=create new data object *)
	write_once : BOOL; (* write permanent memory once *)
	DatObjCreate_01 : DatObjCreate; (* data object create *)
	DatObjInfo_01 : DatObjInfo; (* data object info *)
	DatObjRead_01 : DatObjRead; (* data object read *)
	DatObjWrite_01 : DatObjWrite; (* data object write *)
	ModuleName : STRING[35]; (* module name of object *)
	TON_WritePMEM : TON; (* delay write permanent memory *)
	ulPMPointer : UDINT; (* adress of actual checksum value *)
	ulChecksum : UDINT; (* parameter checksum value *)
	pm_len : UDINT; (* permanent value lenght *)
	ulChecksumOld : UDINT; (* last vlaue of parameter checksum *)
	ulChkValue : UDINT; (* actual value of parameter pointer *)
	pm_id : UDINT; (* permanent value identifier *)
	pm_p : UDINT; (* permanent value pointer *)
END_VAR
VAR CONSTANT
	ERR_NOERROR : UINT := 0;
END_VAR
VAR
	pm_Error : UINT; (* permanent value error *) (* Deleted: pm : ParaMem_typ; permanent memory tags mathias, 22.8.11*)
	xLocalParaCheck : ParaCheckFUB; (*local function instance to check parameter values*)
	TON_BlockMinFileAge : TON; (*waiting time without file write after successful performed write*)
	bBlock_MinFileAge : BOOL := FALSE; (*pause the perm file write after each sucessful write*)
	iPM_WriteCnt : UDINT; (* *) (*old VarName: usPMWriteCnt*)
	TON_WarnDelay : TON := (0);
	bBlock_AutoFileDelete : BOOL := FALSE; (*TRUE will avaod the instant file deletion on detected file errores*)
	DatObjDelete_PermMem : DatObjDelete; (*new V4.13*)
END_VAR
```

### Package Logical/SAFI - SA: SAFI (Sensor Actor Function Interface)


### Data object Logical/SAFI/META_SA (Simple) - SAFI META data module

#### META_SA.dat
```
; *******************************************************************************
; AGGR: Module Meta Data (data module)
;
; This code is confidential and proprietary to the INNIO Company.
; It may not be used in any form, or reproduced in any manner, without the express
; written permission of the INNIO Company.
; Copyright, INNIO Company, 2024
;
; Customized modifications: -
; ------------------------
;
; History:
; -------
; V3.99		06-03-2013	Weitzer, generated for modular software
; V4.00 	31.01.2014	Weitzer, versions changed
; V4.00.4	30-10-2014	Weitzer, correction of sticking at parameter download
;								 correct PV name for coil time 0 power limit
; V4.00.5	28-07-2015	Weitzer, move speed measuring to new task safi_spd
;								 optimize call of misfire command
; V4.03		14-10-2014	Weitzer, PI modified for new CAL Version 7.24
; V4.03.1	10-05-2016	Weitzer, adapt SAFI reset for SAFI1 devices
; V4.04		10-10-2016	Weitzer, add new PI monitoring functionalities
;			27-10-2016	Weitzer, add SAFI FW K7.71, D7.52
;			07-11-2016	Weitzer, improve parameter sending
; V4.05		16-05-2017	Weitzer, add MPM monitoring
;			30-10-2017  Zengerer call for unused interfacet to avoid msg
;			27.07.2017	Messner, CAN Diagnosis Picture added
; V4.5.1	04.12.2017	Weitzer	 SPAX cam monitoring added
;			22-03-2018	Weitzer, Reduce SAFI FW version according to released versions
; V4.05.2	12-03-2017	Weitzer, PI correct current ctr: change reset source to warning
; V4.06.0	05-07-2018	Perktold,activating MPMs also in stop mode if engine should be ready for fast start
; V4.07.0	20-12-2018	Andre,   Added invertion of cross over bit if MORIS rail swapped and shell of valve closure detection
; V4.09.0	27-01-2020	Denk, 	 no warning 3548 “Ignition voltage to high” when selftest is executed
; 			01-04-2020	Andre, 	 Improved PI close detection including PI faults reset and skip fire
; V4.10.0	18-01-2021	Perktold,released dyn spark duration function for all engines
; V4.10.0	28-01-2021	Denk, 	 Alarm deactivation when DGS/WinMOD Simulation is active (3552).
; V4.11.0	16-11-2021	Andre,	 SAFI software reset only if necessary. A3333 if no configuration done bit for 1 min. No A2214 in simulation
;			01.12.2021	Kafka,	 Lambda Controller PBC
;			22-12-2021	Andre,	 Added plausibility check of SAFI measurements. Added type 3 F changes. Added unbalance valve detection
; V4.12.0	25-08-2022	Andre,	 Bug fixes safety loop check and FW version monitoring
;			08-09-2022	Andre,	 Added SEMIC changes.
;			11-11-2022	Andre,	 Added SAFI3/KLS21 changes.
;			05-12-2022	Andre,	 Added 2nd CAN bus card changes.
; V4.13.0	17-10-2023	Andre,	 Fixed issues 1207, 1242, 1244, 1262.
;			08-03-2024	Andre,	 Added KLS21 FW 20.04.
; V4.14.0	10-06-2024	Andre,	 Fixed issue 1492, 1476.
;			07-10-2024	Andre,	 Added activation bit for KLS and DMR parallel mode, enable 2nd CAN bus card for type 9. Fix issue 1587.
;			25-11-2024	Bacci,	 T6 Start procedure with purge start (2024-219): added reset ignition in operation bit
;			27-11-2024	Andre,	 Extended maximum time for skip fire during purge starts with skip fire.
;
; Instructions for use:
; --------------------
; make only changes at the version numbers
;
; Outstandings:
; ------------
; datamodule syntax checker
; (caution: syntax errors here may cause plc runtime errors!)
;
; *******************************************************************************
;
"<META>"
;
; Module ID
"<MODUL>SA</MODUL>"
;
; Module Version (xx.yy.zz.cc)
"<VERSION>04.14.00.00</VERSION>"
;
; Module Basisupdate Version BU (00-99)
"<BASISUPDATE_VERSION>00</BASISUPDATE_VERSION>"
;
; Optional: specify order number for limitated module usage
"<ORDER></ORDER>" ;<!--(optional for restricted customizations; missing statement makes module valid for all orders)-->
;
; Parameter Check <PARAn Name='aAbcdef' MIN='xxx' MAX='yyy' />  (watch for correct spacings and apostrophs!)
"<PARAMETER_CHK>"
"	<PARA1 Name='iEng_Motortype' MIN='208' MAX='920' />"
"	<PARA2 Name='rN_OvrSpeed' MIN='800.0' MAX='2200.0' />"
"	<PARA3 />"
"	<PARA4 />"
"	<PARA5 />"
"</PARAMETER_CHK>"
;
; Permanent Datamodule Filenames<!-- enter filenames for counter and INTERNAL parameter only; filename without extention-->
"<DATAMODULES>" ;<!-- optional; mehrere DATAMODULES erlaubt-->
"	<DATAMODULE>par_SA</DATAMODULE>"
"	<DATAMODULE>CUp_perm</DATAMODULE>"
"</DATAMODULES>"
;
; Dependencies Modules (MMxx.yy.zz.cc)
"<DEPENDENCIES>"
"	<DEPENDENCY MODULE='AB' VERSION='04.00.00.00' />"
"	<DEPENDENCY MODULE='AG' VERSION='04.00.00.00' />"
"	<DEPENDENCY MODULE='CB' VERSION='04.03.00.00' />"
"	<DEPENDENCY MODULE='CH' VERSION='04.03.00.00' />"
"	<DEPENDENCY MODULE='EC' VERSION='04.06.00.00' />"
"	<DEPENDENCY MODULE='GT' VERSION='04.00.00.00' />"
"	<DEPENDENCY MODULE='HA' VERSION='04.12.00.00' />"
"	<DEPENDENCY MODULE='IC' VERSION='04.12.00.00' />"
"	<DEPENDENCY MODULE='IG' VERSION='04.00.00.00' />"
"	<DEPENDENCY MODULE='KN' VERSION='04.11.00.00' />"
"	<DEPENDENCY MODULE='OP' VERSION='04.00.00.00' />"
"	<DEPENDENCY MODULE='PB' VERSION='04.00.00.00' />"
"   <DEPENDENCY VISVERSION='02.13.00.00' />"			; Dependencies Visualization
"</DEPENDENCIES>"
;
; Module function description
"<MODULEFUNCTION>" ;<!-- short overview documentation of module function; add reference to detailed information, if available-->
"	<General>	"
"	CAN communication to SAFI devices. "
"	</General>	"
""
"	<F1 Name='CAN Communication' LastModified='04.00.0.0'>"
"	Manage and monitor CAN communication to SAFI devices.	"
"	</F1>"
"	<F2 Name='Parameter sending' LastModified='04.00.0.0'>"
"	 Send general parameters and operation values to the devices.	"
"	</F2>"
"	<F3 Name='Error handling' LastModified='04.00.0.0'>"
"	 Forward errors from SAFIs to the control system. 	"
"	</F3>"
"	<F4 Name='Ignition' LastModified='04.00.0.0'>"
"	Send ignition parameters and operation values to the devices.	"
"	</F4>"
"	<F5 Name='Knock Detection' LastModified='04.00.0.0'>"
"	Send knocking detection parameters and operation values to the devices.	"
"	</F5>"
"	<F6 Name='High Voltage measurement' LastModified='04.00.0.0'>"
"	Send High voltage measurement parameters and operation values to the devices.	"
"	</F6>"
"	<F7 Name='Pressure based engine control' LastModified='04.00.0.0'>"
"	Send PBC parameters and operation values to the devices.	"
"	</F7>"
"	<F8 Name='Port injection' LastModified='04.00.0.0'>"
"	Send port injection parameters and operation values to the devices.	"
"	</F8>"
"	<F9 Name='Valve closure detection' LastModified='04.07.0.0'>"
"	Detect valve closure noise and timing.	"
"	</F9>"
"	<Info>"
"	no furhter information	"
"	</Info>"
""
"	<Customized LastModified='04.00.0.1'>	"
"	- Nothing "
"	</Customized>	"
""
"</MODULEFUNCTION>"
;
"</META>"
```
